C05458=1063.353,412.213,382.958,175.388,37.481,157.115
C05459=1063.360,412.459,382.914,175.394,37.490,157.117
C05460=1063.368,412.705,382.870,175.401,37.500,157.119
C05461=1063.377,412.951,382.826,175.409,37.509,157.122
C05462=1063.386,413.197,382.781,175.416,37.519,157.124
C05463=1063.394,413.443,382.737,175.423,37.528,157.127
C05464=1063.402,413.689,382.693,175.429,37.537,157.129
C05465=1063.411,413.935,382.648,175.436,37.547,157.131
C05466=1063.419,414.181,382.604,175.444,37.556,157.134
C05467=1063.427,414.426,382.559,175.451,37.566,157.136
C05468=1063.438,414.737,382.503,175.459,37.578,157.140
C05469=1063.448,415.046,382.447,175.468,37.590,157.143
C05470=1063.459,415.356,382.391,175.478,37.602,157.146
C05471=1063.469,415.665,382.334,175.486,37.614,157.149
C05472=1063.477,415.911,382.289,175.494,37.624,157.152
C05473=1063.486,416.157,382.245,175.501,37.634,157.154
C05474=1063.494,416.402,382.200,175.508,37.643,157.157
C05475=1063.503,416.648,382.155,175.516,37.653,157.159
C05476=1063.511,416.894,382.110,175.523,37.663,157.162
C05477=1063.520,417.140,382.066,175.530,37.673,157.164
C05478=1063.528,417.385,382.021,175.538,37.683,157.167
C05479=1063.537,417.632,381.976,175.545,37.692,157.170
C05480=1063.545,417.877,381.931,175.553,37.702,157.172
C05481=1063.553,418.123,381.885,175.560,37.712,157.175
C05482=1063.561,418.369,381.840,175.567,37.722,157.177
C05483=1063.570,418.614,381.795,175.575,37.732,157.180
C05484=1063.579,418.860,381.750,175.582,37.742,157.183
C05485=1063.587,419.106,381.705,175.590,37.752,157.185
C05486=1063.596,419.352,381.660,175.597,37.762,157.188
C05487=1063.605,419.597,381.615,175.605,37.772,157.191
C05488=1063.613,419.843,381.569,175.612,37.782,157.193
C05489=1063.622,420.089,381.523,175.620,37.792,157.196
C05490=1063.631,420.335,381.478,175.627,37.803,157.199
C05491=1063.640,420.581,381.433,175.635,37.813,157.201
C05492=1063.648,420.826,381.387,175.643,37.823,157.204
C05493=1063.657,421.072,381.341,175.650,37.833,157.207
C05494=1063.665,421.318,381.296,175.658,37.843,157.210
C05495=1063.673,421.563,381.250,175.665,37.854,157.212
C05496=1063.682,421.808,381.204,175.674,37.864,157.215
C05497=1063.691,422.054,381.158,175.681,37.875,157.218
C05498=1063.700,422.300,381.113,175.689,37.885,157.221
C05499=1063.708,422.546,381.066,175.697,37.896,157.224
C05500=1063.717,422.791,381.021,175.704,37.906,157.226
C05501=1063.726,423.037,380.976,175.713,37.917,157.229
C05502=1063.734,423.282,380.929,175.721,37.927,157.232
C05503=1063.743,423.528,380.883,175.728,37.938,157.235
C05504=1063.752,423.774,380.837,175.736,37.948,157.238
C05505=1063.761,424.019,380.791,175.745,37.959,157.241
C05506=1063.769,424.265,380.745,175.753,37.970,157.244
C05507=1063.778,424.510,380.698,175.760,37.981,157.246
C05508=1063.787,424.756,380.652,175.768,37.991,157.249
C05509=1063.796,425.001,380.606,175.777,38.002,157.252
C05510=1063.804,425.247,380.560,175.785,38.013,157.255
C05511=1063.814,425.492,380.513,175.793,38.024,157.258
C05512=1063.822,425.738,380.467,175.801,38.034,157.261
C05513=1063.832,425.983,380.421,175.809,38.045,157.264
C05514=1063.840,426.229,380.375,175.817,38.056,157.267
C05515=1063.849,426.474,380.328,175.826,38.067,157.270
C05516=1063.858,426.720,380.282,175.834,38.078,157.273
C05517=1063.868,426.966,380.235,175.843,38.089,157.276
C05518=1063.876,427.211,380.188,175.851,38.100,157.279
C05519=1063.885,427.456,380.141,175.860,38.111,157.282
C05520=1063.893,427.702,380.094,175.868,38.122,157.285
C05521=1063.903,427.947,380.048,175.875,38.134,157.288
C05522=1063.912,428.192,380.001,175.884,38.145,157.291
C05523=1063.921,428.438,379.954,175.893,38.156,157.294
C05524=1063.933,428.768,379.890,175.904,38.171,157.298
C05525=1063.945,429.097,379.828,175.916,38.186,157.302
C05526=1063.957,429.427,379.764,175.928,38.202,157.307
C05527=1063.969,429.757,379.701,175.939,38.217,157.311
C05528=1063.978,430.001,379.654,175.948,38.229,157.314
C05529=1063.988,430.247,379.607,175.956,38.240,157.317
C05530=1063.996,430.492,379.560,175.965,38.251,157.320
C05531=1064.006,430.738,379.512,175.974,38.263,157.323
C05532=1064.015,430.983,379.464,175.982,38.274,157.327
C05533=1064.023,431.228,379.418,175.992,38.286,157.330
C05534=1064.033,431.474,379.370,176.001,38.298,157.333
C05535=1064.042,431.719,379.322,176.009,38.310,157.336
C05536=1064.051,431.964,379.275,176.018,38.322,157.340
C05537=1064.060,432.209,379.227,176.027,38.334,157.343
C05538=1064.069,432.455,379.179,176.036,38.345,157.346
C05539=1064.078,432.700,379.132,176.045,38.357,157.350
C05540=1064.088,432.945,379.083,176.054,38.369,157.353
C05541=1064.097,433.190,379.036,176.063,38.381,157.356
C05542=1064.106,433.435,378.988,176.072,38.393,157.359
C05543=1064.116,433.681,378.940,176.082,38.405,157.363
C05544=1064.125,433.925,378.892,176.090,38.417,157.366
C05545=1064.134,434.171,378.844,176.099,38.429,157.369
C05546=1064.144,434.416,378.797,176.109,38.441,157.373
C05547=1064.153,434.660,378.748,176.118,38.454,157.376
C05548=1064.162,434.906,378.701,176.128,38.466,157.380
C05549=1064.172,435.151,378.652,176.137,38.478,157.383
C05550=1064.180,435.396,378.604,176.146,38.490,157.387
C05551=1064.190,435.641,378.556,176.156,38.503,157.390
C05552=1064.200,435.886,378.507,176.165,38.515,157.394
C05553=1064.209,436.132,378.459,176.175,38.527,157.397
C05554=1064.219,436.377,378.411,176.184,38.539,157.400
C05555=1064.229,436.622,378.362,176.194,38.552,157.404
C05556=1064.239,436.867,378.314,176.203,38.564,157.407
C05557=1064.248,437.112,378.265,176.213,38.577,157.411
C05558=1064.257,437.356,378.216,176.223,38.590,157.415
C05559=1064.266,437.601,378.168,176.232,38.602,157.418
C05560=1064.277,437.847,378.119,176.242,38.615,157.422
C05561=1064.287,438.092,378.070,176.251,38.627,157.425
C05562=1064.296,438.337,378.022,176.261,38.640,157.429
C05563=1064.305,438.582,377.973,176.272,38.653,157.433
C05564=1064.315,438.826,377.924,176.281,38.666,157.436
C05565=1064.325,439.071,377.875,176.291,38.679,157.440
C05566=1064.334,439.317,377.826,176.301,38.692,157.444
C05567=1064.344,439.561,377.777,176.310,38.705,157.447
C05568=1064.353,439.806,377.727,176.321,38.718,157.451
C05569=1064.363,440.051,377.678,176.331,38.731,157.455
C05570=1064.373,440.296,377.630,176.341,38.743,157.458
C05571=1064.383,440.541,377.580,176.352,38.757,157.462
C05572=1064.393,440.786,377.531,176.361,38.770,157.466
C05573=1064.402,441.031,377.481,176.372,38.783,157.470
C05574=1064.412,441.275,377.432,176.382,38.797,157.474
C05575=1064.422,441.520,377.382,176.392,38.810,157.477
C05576=1064.432,441.765,377.332,176.403,38.823,157.481
C05577=1064.441,442.010,377.283,176.413,38.836,157.485
C05578=1064.451,442.254,377.234,176.424,38.850,157.489
C05579=1064.461,442.500,377.184,176.434,38.864,157.493
C05580=1064.477,442.869,377.108,176.449,38.884,157.499
C05581=1064.491,443.240,377.033,176.466,38.904,157.505
C05582=1064.507,443.611,376.957,176.482,38.925,157.511
C05583=1064.522,443.980,376.881,176.498,38.946,157.517
C05584=1064.532,444.225,376.832,176.508,38.960,157.521
C05585=1064.542,444.470,376.782,176.519,38.974,157.525
C05586=1064.551,444.714,376.731,176.531,38.987,157.529
C05587=1064.562,444.959,376.682,176.542,39.001,157.533
C05588=1064.572,445.204,376.631,176.552,39.015,157.537
C05589=1064.582,445.448,376.580,176.563,39.029,157.541
C05590=1064.592,445.693,376.531,176.574,39.043,157.545
C05591=1064.603,445.938,376.480,176.586,39.057,157.549
C05592=1064.612,446.182,376.429,176.597,39.072,157.554
C05593=1064.623,446.427,376.378,176.607,39.086,157.558
C05594=1064.633,446.671,376.328,176.619,39.100,157.562
C05595=1064.644,446.916,376.277,176.630,39.114,157.566
C05596=1064.653,447.160,376.226,176.641,39.129,157.570
C05597=1064.664,447.403,376.176,176.653,39.143,157.575
C05598=1064.674,447.647,376.126,176.664,39.158,157.579
C05599=1064.685,447.891,376.075,176.676,39.172,157.583
C05600=1064.697,448.135,376.026,176.687,39.186,157.587
C05601=1064.710,448.379,375.977,176.699,39.199,157.591
C05602=1064.724,448.624,375.929,176.710,39.213,157.595
C05603=1064.739,448.868,375.882,176.722,39.226,157.599
C05604=1064.755,449.113,375.834,176.734,39.238,157.603
C05605=1064.773,449.358,375.788,176.746,39.251,157.607
C05606=1064.791,449.603,375.742,176.758,39.263,157.610
C05607=1064.810,449.849,375.697,176.768,39.275,157.614
C05608=1064.471,449.855,375.431,176.760,39.399,157.648
C05609=1064.452,449.610,375.475,176.748,39.387,157.644
C05610=1064.434,449.364,375.521,176.737,39.375,157.640
C05611=1064.417,449.119,375.566,176.725,39.362,157.637
C05612=1064.401,448.875,375.613,176.713,39.350,157.633
C05613=1064.386,448.629,375.661,176.701,39.337,157.629
C05614=1064.371,448.385,375.710,176.689,39.324,157.625
C05615=1064.358,448.141,375.758,176.678,39.310,157.621
C05616=1064.345,447.897,375.807,176.666,39.296,157.617
C05617=1064.334,447.653,375.858,176.654,39.282,157.612
C05618=1064.324,447.409,375.908,176.643,39.268,157.608
C05619=1064.313,447.165,375.959,176.631,39.254,157.604
C05620=1064.303,446.921,376.009,176.620,39.240,157.600
C05621=1064.293,446.677,376.060,176.609,39.225,157.595
C05622=1064.283,446.433,376.111,176.597,39.211,157.591
C05623=1064.272,446.188,376.161,176.586,39.197,157.587
C05624=1064.262,445.943,376.212,176.575,39.183,157.583
C05625=1064.252,445.699,376.263,176.564,39.169,157.579
C05626=1064.242,445.455,376.313,176.553,39.155,157.575
C05627=1064.231,445.210,376.364,176.542,39.141,157.571
C05628=1064.221,444.965,376.414,176.531,39.127,157.566
C05629=1064.211,444.721,376.464,176.519,39.113,157.562
C05630=1064.201,444.476,376.514,176.508,39.099,157.558
C05631=1064.190,444.231,376.565,176.498,39.085,157.554
C05632=1064.181,443.986,376.615,176.487,39.071,157.550
C05633=1064.167,443.636,376.687,176.472,39.052,157.544
C05634=1064.152,443.284,376.759,176.456,39.032,157.539
C05635=1064.138,442.934,376.830,176.441,39.012,157.533
C05636=1064.123,442.583,376.902,176.425,38.993,157.527
C05637=1064.113,442.337,376.952,176.414,38.980,157.523
C05638=1064.103,442.093,377.001,176.404,38.967,157.520
C05639=1064.094,441.848,377.051,176.394,38.953,157.516
C05640=1064.083,441.603,377.100,176.384,38.940,157.512
C05641=1064.074,441.358,377.150,176.373,38.926,157.508
C05642=1064.064,441.114,377.200,176.363,38.913,157.504
C05643=1064.055,440.869,377.249,176.352,38.900,157.500
C05644=1064.044,440.624,377.298,176.342,38.887,157.497
C05645=1064.035,440.379,377.348,176.332,38.874,157.493
C05646=1064.025,440.135,377.397,176.321,38.861,157.489
C05647=1064.016,439.890,377.446,176.312,38.847,157.485
C05648=1064.005,439.644,377.496,176.302,38.835,157.482
C05649=1063.995,439.399,377.545,176.291,38.822,157.478
C05650=1063.986,439.155,377.594,176.281,38.809,157.474
C05651=1063.976,438.910,377.643,176.272,38.796,157.470
C05652=1063.966,438.665,377.691,176.261,38.783,157.467
C05653=1063.957,438.420,377.741,176.251,38.770,157.463
C05654=1063.947,438.175,377.790,176.242,38.758,157.460
C05655=1063.938,437.930,377.838,176.232,38.745,157.456
C05656=1063.928,437.685,377.887,176.221,38.732,157.452
C05657=1063.919,437.440,377.936,176.212,38.720,157.449
C05658=1063.909,437.195,377.985,176.202,38.707,157.445
C05659=1063.899,436.950,378.033,176.193,38.695,157.442
C05660=1063.890,436.705,378.082,176.183,38.682,157.438
C05661=1063.880,436.460,378.130,176.173,38.670,157.435
C05662=1063.870,436.215,378.179,176.164,38.658,157.431
C05663=1063.860,435.970,378.227,176.154,38.645,157.428
C05664=1063.851,435.725,378.276,176.145,38.633,157.424
C05665=1063.842,435.479,378.324,176.135,38.620,157.421
C05666=1063.833,435.235,378.372,176.126,38.608,157.417
C05667=1063.823,434.990,378.421,176.117,38.596,157.414
C05668=1063.813,434.744,378.469,176.107,38.584,157.410
C05669=1063.804,434.500,378.517,176.098,38.572,157.407
C05670=1063.795,434.255,378.565,176.088,38.560,157.404
C05671=1063.785,434.010,378.613,176.079,38.547,157.400
C05672=1063.776,433.764,378.661,176.070,38.536,157.397
C05673=1063.767,433.519,378.708,176.060,38.523,157.393
C05674=1063.757,433.274,378.757,176.051,38.512,157.390
C05675=1063.748,433.029,378.805,176.042,38.500,157.387
C05676=1063.739,432.784,378.852,176.032,38.488,157.383
C05677=1063.729,432.538,378.900,176.024,38.476,157.380
C05678=1063.720,432.293,378.947,176.015,38.464,157.377
C05679=1063.711,432.048,378.996,176.006,38.452,157.373
C05680=1063.702,431.803,379.043,175.997,38.440,157.370
C05681=1063.692,431.558,379.091,175.987,38.429,157.367
C05682=1063.683,431.313,379.139,175.979,38.417,157.364
C05683=1063.674,431.067,379.186,175.970,38.405,157.360
C05684=1063.665,430.822,379.233,175.961,38.394,157.357
C05685=1063.656,430.576,379.281,175.953,38.382,157.354
C05686=1063.647,430.331,379.328,175.944,38.371,157.351
C05687=1063.638,430.086,379.376,175.934,38.360,157.348
C05688=1063.629,429.840,379.423,175.925,38.348,157.345
C05689=1063.616,429.509,379.487,175.914,38.332,157.340
C05690=1063.605,429.178,379.550,175.902,38.317,157.336
C05691=1063.592,428.846,379.614,175.891,38.302,157.332
C05692=1063.579,428.514,379.677,175.879,38.287,157.328
C05693=1063.570,428.269,379.725,175.871,38.276,157.325
C05694=1063.562,428.024,379.771,175.862,38.264,157.322
C05695=1063.553,427.778,379.818,175.854,38.253,157.319
C05696=1063.543,427.533,379.865,175.845,38.242,157.315
C05697=1063.535,427.287,379.912,175.837,38.231,157.312
C05698=1063.526,427.042,379.959,175.828,38.220,157.309
C05699=1063.517,426.796,380.005,175.820,38.209,157.306
C05700=1063.508,426.551,380.052,175.811,38.198,157.303
C05701=1063.499,426.305,380.099,175.803,38.187,157.300
C05702=1063.490,426.060,380.145,175.794,38.176,157.297
C05703=1063.481,425.814,380.191,175.787,38.165,157.294
C05704=1063.472,425.569,380.238,175.779,38.154,157.292
C05705=1063.463,425.323,380.284,175.770,38.144,157.289
C05706=1063.454,425.078,380.330,175.762,38.133,157.286
C05707=1063.446,424.833,380.377,175.753,38.122,157.283
C05708=1063.437,424.587,380.423,175.745,38.111,157.280
C05709=1063.428,424.341,380.469,175.738,38.100,157.277
C05710=1063.419,424.096,380.515,175.729,38.090,157.274
C05711=1063.410,423.850,380.561,175.721,38.079,157.271
C05712=1063.401,423.605,380.608,175.713,38.069,157.268
C05713=1063.392,423.360,380.654,175.706,38.058,157.265
C05714=1063.384,423.113,380.700,175.697,38.047,157.263
C05715=1063.374,422.868,380.746,175.689,38.037,157.260
C05716=1063.366,422.622,380.792,175.682,38.027,157.257
C05717=1063.357,422.376,380.837,175.673,38.016,157.254
C05718=1063.349,422.131,380.884,175.665,38.006,157.251
C05719=1063.340,421.886,380.929,175.658,37.995,157.248
C05720=1063.331,421.640,380.975,175.650,37.985,157.246
C05721=1063.323,421.394,381.021,175.643,37.975,157.243
C05722=1063.314,421.149,381.067,175.634,37.964,157.240
C05723=1063.306,420.903,381.112,175.626,37.954,157.237
C05724=1063.297,420.657,381.158,175.619,37.944,157.235
C05725=1063.288,420.411,381.203,175.611,37.934,157.232
C05726=1063.280,420.165,381.249,175.604,37.924,157.229
C05727=1063.272,419.920,381.294,175.596,37.913,157.227
C05728=1063.263,419.674,381.340,175.589,37.903,157.224
C05729=1063.254,419.429,381.385,175.580,37.893,157.221
C05730=1063.245,419.183,381.430,175.573,37.883,157.219
C05731=1063.236,418.938,381.476,175.565,37.873,157.216
C05732=1063.228,418.691,381.522,175.558,37.863,157.213
C05733=1063.220,418.446,381.566,175.550,37.853,157.210
C05734=1063.211,418.200,381.611,175.543,37.844,157.208
C05735=1063.202,417.954,381.657,175.535,37.834,157.205
C05736=1063.194,417.709,381.702,175.528,37.824,157.203
C05737=1063.185,417.462,381.746,175.520,37.814,157.200
C05738=1063.177,417.217,381.792,175.513,37.804,157.197
C05739=1063.168,416.971,381.836,175.506,37.794,157.195
C05740=1063.160,416.725,381.882,175.498,37.784,157.192
C05741=1063.152,416.479,381.927,175.491,37.775,157.190
C05742=1063.143,416.234,381.972,175.484,37.765,157.187
C05743=1063.135,415.987,382.016,175.476,37.755,157.185
C05744=1063.126,415.742,382.061,175.469,37.745,157.182
C05745=1063.115,415.431,382.118,175.460,37.733,157.179
C05746=1063.104,415.119,382.175,175.451,37.721,157.176
C05747=1063.095,414.808,382.231,175.442,37.709,157.172
C05748=1063.084,414.496,382.288,175.432,37.697,157.169
C05749=1063.076,414.251,382.332,175.426,37.687,157.167
C05750=1063.067,414.004,382.377,175.419,37.678,157.164
C05751=1063.059,413.759,382.421,175.411,37.668,157.162
C05752=1063.051,413.513,382.465,175.404,37.659,157.159
C05753=1063.042,413.267,382.510,175.397,37.650,157.157
C05754=1063.034,413.021,382.554,175.390,37.640,157.154
C05755=1063.025,412.775,382.598,175.384,37.631,157.152
C05756=1063.016,412.529,382.642,175.376,37.622,157.150
C05757=1063.008,412.283,382.687,175.369,37.613,157.147
C05758=1063.000,412.037,382.731,175.362,37.603,157.145
C05759=1062.992,411.792,382.775,175.355,37.594,157.142
C05760=1062.983,411.545,382.819,175.349,37.585,157.140
C05761=1062.975,411.299,382.863,175.342,37.576,157.138
C05762=1062.967,411.053,382.907,175.335,37.567,157.135
C05763=1062.958,410.807,382.950,175.327,37.558,157.133
C05764=1062.950,410.562,382.995,175.321,37.549,157.131
C05765=1062.942,410.316,383.039,175.314,37.540,157.128
C05766=1062.934,410.070,383.083,175.307,37.531,157.126
C05767=1062.926,409.824,383.126,175.300,37.522,157.124
C05768=1062.917,409.577,383.170,175.294,37.513,157.121
C05769=1062.909,409.331,383.215,175.287,37.504,157.119
C05770=1062.901,409.085,383.258,175.280,37.495,157.117
C05771=1062.893,408.839,383.301,175.274,37.486,157.114
C05772=1062.885,408.593,383.346,175.267,37.477,157.112
C05773=1062.876,408.347,383.389,175.260,37.468,157.110
C05774=1062.869,408.101,383.432,175.254,37.459,157.107
C05775=1062.861,407.856,383.476,175.247,37.450,157.105
C05776=1062.853,407.610,383.519,175.240,37.441,157.103
C05777=1062.845,407.363,383.563,175.234,37.432,157.101
C05778=1062.837,407.117,383.607,175.227,37.424,157.098
C05779=1062.829,406.871,383.650,175.220,37.415,157.096
C05780=1062.821,406.625,383.694,175.214,37.406,157.094
C05781=1062.813,406.379,383.738,175.208,37.398,157.092
C05782=1062.805,406.133,383.780,175.202,37.389,157.089
C05783=1062.797,405.887,383.824,175.195,37.380,157.087
C05784=1062.789,405.641,383.867,175.188,37.372,157.085
C05785=1062.781,405.395,383.911,175.182,37.363,157.083
C05786=1062.773,405.148,383.953,175.175,37.355,157.081
C05787=1062.765,404.902,383.997,175.169,37.346,157.078
C05788=1062.757,404.656,384.039,175.162,37.337,157.076
C05789=1062.749,404.410,384.083,175.157,37.329,157.074
C05790=1062.741,404.164,384.126,175.150,37.320,157.072
C05791=1062.734,403.917,384.168,175.144,37.312,157.070
C05792=1062.725,403.671,384.211,175.137,37.303,157.068
C05793=1062.717,403.425,384.254,175.131,37.295,157.066
C05794=1062.709,403.178,384.297,175.125,37.287,157.063
C05795=1062.702,402.933,384.340,175.119,37.279,157.061
C05796=1062.693,402.687,384.383,175.112,37.270,157.059
C05797=1062.686,402.440,384.426,175.106,37.261,157.057
C05798=1062.678,402.195,384.469,175.099,37.253,157.055
C05799=1062.669,401.948,384.511,175.094,37.245,157.053
C05800=1062.661,401.702,384.554,175.087,37.237,157.051
C05801=1062.652,401.395,384.606,175.079,37.227,157.048
C05802=1062.642,401.089,384.659,175.072,37.216,157.046
C05803=1062.632,400.783,384.713,175.064,37.206,157.043
C05804=1062.622,400.476,384.765,175.056,37.196,157.040
C05805=1062.615,400.230,384.807,175.051,37.188,157.038
C05806=1062.606,399.984,384.850,175.044,37.180,157.036
C05807=1062.599,399.738,384.893,175.038,37.172,157.034
C05808=1062.591,399.491,384.935,175.033,37.164,157.032
C05809=1062.584,399.245,384.977,175.026,37.156,157.030
C05810=1062.575,398.999,385.019,175.020,37.148,157.028
C05811=1062.568,398.753,385.061,175.014,37.140,157.026
C05812=1062.560,398.506,385.104,175.008,37.132,157.024
C05813=1062.552,398.261,385.146,175.002,37.124,157.022
C05814=1062.545,398.014,385.189,174.996,37.116,157.020
C05815=1062.537,397.768,385.231,174.990,37.108,157.018
C05816=1062.529,397.521,385.272,174.985,37.100,157.016
C05817=1062.522,397.275,385.314,174.978,37.092,157.014
C05818=1062.513,397.028,385.357,174.972,37.085,157.012
C05819=1062.506,396.782,385.398,174.967,37.077,157.010
C05820=1062.498,396.537,385.440,174.960,37.069,157.009
C05821=1062.490,396.290,385.483,174.955,37.061,157.007
C05822=1062.483,396.043,385.524,174.949,37.053,157.005
C05823=1062.474,395.798,385.565,174.943,37.046,157.003
C05824=1062.467,395.552,385.607,174.937,37.038,157.001
C05825=1062.459,395.305,385.650,174.931,37.030,156.999
C05826=1062.451,395.058,385.691,174.926,37.023,156.997
C05827=1062.444,394.812,385.733,174.919,37.014,156.995
C05828=1062.436,394.566,385.775,174.914,37.007,156.993
C05829=1062.428,394.319,385.816,174.908,36.999,156.991
C05830=1062.421,394.073,385.858,174.902,36.992,156.989
C05831=1062.413,393.827,385.899,174.896,36.984,156.987
C05832=1062.406,393.581,385.941,174.891,36.977,156.986
C05833=1062.398,393.334,385.982,174.885,36.969,156.984
C05834=1062.391,393.088,386.023,174.880,36.961,156.982
C05835=1062.383,392.842,386.065,174.873,36.954,156.980
C05836=1062.376,392.595,386.106,174.868,36.946,156.978
C05837=1062.367,392.349,386.148,174.862,36.939,156.976
C05838=1062.359,392.102,386.189,174.857,36.932,156.974
C05839=1062.352,391.856,386.231,174.850,36.924,156.973
C05840=1062.345,391.609,386.272,174.845,36.916,156.971
C05841=1062.337,391.363,386.313,174.840,36.909,156.969
C05842=1062.329,391.117,386.354,174.834,36.902,156.967
C05843=1062.322,390.870,386.396,174.829,36.895,156.965
C05844=1062.314,390.624,386.436,174.823,36.887,156.963
C05845=1062.307,390.377,386.478,174.817,36.880,156.962
C05846=1062.299,390.131,386.519,174.811,36.872,156.960
C05847=1062.291,389.884,386.559,174.806,36.865,156.958
C05848=1062.284,389.638,386.601,174.801,36.858,156.956
C05849=1062.276,389.391,386.641,174.795,36.851,156.955
C05850=1062.269,389.145,386.682,174.790,36.844,156.953
C05851=1062.261,388.899,386.723,174.784,36.836,156.951
C05852=1062.254,388.653,386.764,174.778,36.829,156.949
C05853=1062.246,388.406,386.805,174.773,36.822,156.947
C05854=1062.239,388.160,386.846,174.767,36.815,156.946
C05855=1062.231,387.914,386.886,174.762,36.808,156.944
C05856=1062.223,387.667,386.926,174.757,36.801,156.942
C05857=1062.214,387.377,386.975,174.751,36.792,156.940
C05858=1062.205,387.088,387.023,174.743,36.784,156.938
C05859=1062.196,386.798,387.070,174.737,36.775,156.936
C05860=1062.188,386.508,387.118,174.731,36.767,156.934
C05861=1062.180,386.262,387.159,174.726,36.760,156.932
C05862=1062.173,386.015,387.199,174.721,36.753,156.931
C05863=1062.165,385.769,387.240,174.714,36.746,156.929
C05864=1062.158,385.522,387.280,174.709,36.739,156.927
C05865=1062.150,385.275,387.321,174.704,36.732,156.926
C05866=1062.143,385.029,387.360,174.699,36.725,156.924
C05867=1062.136,384.783,387.402,174.693,36.718,156.922
C05868=1062.128,384.536,387.441,174.688,36.712,156.921
C05869=1062.120,384.289,387.482,174.683,36.704,156.919
C05870=1062.114,384.043,387.522,174.678,36.697,156.917
C05871=1062.106,383.796,387.562,174.672,36.691,156.916
C05872=1062.099,383.549,387.603,174.667,36.684,156.914
C05873=1062.092,383.303,387.643,174.662,36.677,156.912
C05874=1062.084,383.056,387.683,174.657,36.670,156.911
C05875=1062.077,382.810,387.724,174.651,36.663,156.909
C05876=1062.070,382.564,387.764,174.646,36.656,156.907
C05877=1062.062,382.317,387.804,174.641,36.650,156.906
C05878=1062.056,382.070,387.844,174.636,36.643,156.904
C05879=1062.048,381.824,387.884,174.631,36.636,156.902
C05880=1062.040,381.578,387.924,174.626,36.629,156.901
C05881=1062.033,381.330,387.964,174.620,36.622,156.899
C05882=1062.026,381.084,388.004,174.615,36.616,156.897
C05883=1062.019,380.837,388.044,174.610,36.609,156.896
C05884=1062.011,380.591,388.083,174.605,36.602,156.894
C05885=1062.004,380.344,388.124,174.600,36.596,156.893
C05886=1061.997,380.097,388.164,174.595,36.589,156.891
C05887=1061.990,379.851,388.203,174.589,36.583,156.890
C05888=1061.982,379.604,388.243,174.584,36.576,156.888
C05889=1061.975,379.358,388.283,174.579,36.569,156.886
C05890=1061.967,379.111,388.323,174.574,36.563,156.885
C05891=1061.960,378.864,388.362,174.569,36.556,156.883
C05892=1061.953,378.617,388.402,174.564,36.550,156.882
C05893=1061.945,378.371,388.441,174.559,36.543,156.880
C05894=1061.938,378.124,388.481,174.553,36.536,156.878
C05895=1061.931,377.877,388.520,174.549,36.530,156.877
C05896=1061.923,377.630,388.560,174.544,36.524,156.875
C05897=1061.916,377.384,388.599,174.539,36.517,156.874
C05898=1061.909,377.137,388.638,174.534,36.511,156.872
C05899=1061.902,376.890,388.678,174.529,36.504,156.871
C05900=1061.894,376.644,388.718,174.524,36.498,156.869
C05901=1061.887,376.397,388.757,174.519,36.491,156.868
C05902=1061.880,376.150,388.796,174.514,36.485,156.866
C05903=1061.873,375.904,388.835,174.509,36.479,156.865
C05904=1061.865,375.657,388.875,174.504,36.472,156.863
C05905=1061.859,375.410,388.914,174.499,36.466,156.862
C05906=1061.851,375.164,388.954,174.495,36.459,156.860
C05907=1061.844,374.916,388.993,174.490,36.453,156.859
C05908=1061.837,374.670,389.032,174.485,36.446,156.857
C05909=1061.830,374.423,389.071,174.480,36.440,156.856
C05910=1061.823,374.176,389.110,174.475,36.434,156.854
C05911=1061.816,373.929,389.150,174.470,36.428,156.853
C05912=1061.809,373.682,389.189,174.465,36.422,156.851
C05913=1061.801,373.423,389.229,174.459,36.415,156.850
C05914=1061.794,373.166,389.271,174.455,36.408,156.848
C05915=1061.786,372.907,389.311,174.450,36.402,156.846
C05916=1061.779,372.648,389.352,174.445,36.395,156.845
C05917=1061.773,372.411,389.389,174.440,36.389,156.843
C05918=1061.765,372.175,389.427,174.435,36.383,156.842
C05919=1061.758,371.938,389.464,174.431,36.377,156.841
C05920=1061.751,371.701,389.501,174.427,36.372,156.839
C05921=1061.744,371.455,389.539,174.422,36.365,156.838
C05922=1061.737,371.208,389.578,174.417,36.359,156.836
C05923=1061.730,370.962,389.618,174.412,36.353,156.835
C05924=1061.722,370.715,389.656,174.407,36.347,156.834
C05925=1061.715,370.467,389.695,174.402,36.341,156.832
C05926=1061.708,370.220,389.733,174.398,36.335,156.831
C05927=1061.701,369.974,389.772,174.393,36.329,156.829
C05928=1061.694,369.727,389.810,174.388,36.323,156.828
C05929=1061.687,369.480,389.849,174.383,36.317,156.827
C05930=1061.680,369.234,389.888,174.378,36.311,156.825
C05931=1061.673,368.987,389.926,174.374,36.305,156.824
C05932=1061.665,368.740,389.965,174.369,36.298,156.822
C05933=1061.659,368.493,390.003,174.365,36.293,156.821
C05934=1061.651,368.246,390.041,174.360,36.287,156.820
C05935=1061.644,367.999,390.080,174.355,36.281,156.818
C05936=1061.637,367.752,390.119,174.351,36.274,156.817
C05937=1061.630,367.505,390.157,174.346,36.269,156.815
C05938=1061.623,367.258,390.195,174.341,36.263,156.814
C05939=1061.615,367.011,390.234,174.336,36.257,156.812
C05940=1061.609,366.764,390.272,174.332,36.251,156.811
C05941=1061.602,366.517,390.311,174.328,36.245,156.810
C05942=1061.595,366.270,390.348,174.323,36.239,156.808
C05943=1061.588,366.023,390.387,174.318,36.233,156.807
C05944=1061.581,365.776,390.424,174.313,36.227,156.806
C05945=1061.575,365.530,390.463,174.309,36.222,156.804
C05946=1061.567,365.283,390.500,174.304,36.215,156.803
C05947=1061.561,365.036,390.539,174.300,36.210,156.802
C05948=1061.554,364.789,390.577,174.295,36.204,156.800
C05949=1061.547,364.542,390.616,174.291,36.198,156.799
C05950=1061.540,364.295,390.654,174.286,36.192,156.797
C05951=1061.532,364.048,390.692,174.281,36.186,156.796
C05952=1061.525,363.801,390.730,174.277,36.181,156.795
C05953=1061.519,363.554,390.768,174.273,36.175,156.793
C05954=1061.511,363.306,390.805,174.268,36.169,156.792
C05955=1061.505,363.061,390.843,174.263,36.163,156.791
C05956=1061.498,362.813,390.881,174.259,36.158,156.790
C05957=1061.491,362.566,390.919,174.255,36.152,156.788
C05958=1061.484,362.319,390.956,174.250,36.146,156.787
C05959=1061.477,362.071,390.994,174.245,36.140,156.786
C05960=1061.469,361.825,391.033,174.241,36.135,156.784
C05961=1061.462,361.578,391.070,174.237,36.129,156.783
C05962=1061.456,361.331,391.108,174.232,36.124,156.782
C05963=1061.449,361.084,391.145,174.228,36.118,156.780
C05964=1061.442,360.837,391.183,174.223,36.112,156.779
C05965=1061.435,360.590,391.220,174.219,36.107,156.778
C05966=1061.427,360.343,391.258,174.215,36.101,156.777
C05967=1061.421,360.096,391.296,174.210,36.096,156.775
C05968=1061.414,359.849,391.333,174.205,36.090,156.774
C05969=1061.407,359.597,391.372,174.202,36.084,156.773
C05970=1061.400,359.347,391.409,174.197,36.079,156.771
C05971=1061.393,359.095,391.448,174.192,36.073,156.770
C05972=1061.386,358.845,391.486,174.187,36.067,156.769
C05973=1061.379,358.597,391.523,174.184,36.062,156.768
C05974=1061.372,358.350,391.560,174.179,36.056,156.766
C05975=1061.365,358.103,391.598,174.174,36.051,156.765
C05976=1061.358,357.857,391.635,174.171,36.045,156.764
C05977=1061.351,357.609,391.672,174.166,36.039,156.762
C05978=1061.345,357.361,391.710,174.161,36.034,156.761
C05979=1061.338,357.115,391.747,174.157,36.029,156.760
C05980=1061.331,356.868,391.785,174.153,36.023,156.759
C05981=1061.324,356.620,391.821,174.148,36.018,156.758
C05982=1061.317,356.374,391.859,174.144,36.012,156.756
C05983=1061.310,356.126,391.896,174.140,36.007,156.755
C05984=1061.303,355.879,391.933,174.136,36.002,156.754
C05985=1061.296,355.632,391.970,174.131,35.996,156.752
C05986=1061.290,355.385,392.007,174.127,35.991,156.751
C05987=1061.283,355.138,392.044,174.123,35.985,156.750
C05988=1061.276,354.890,392.081,174.119,35.980,156.749
C05989=1061.269,354.643,392.118,174.114,35.975,156.748
C05990=1061.262,354.396,392.155,174.110,35.969,156.746
C05991=1061.255,354.149,392.192,174.106,35.964,156.745
C05992=1061.249,353.902,392.229,174.101,35.958,156.744
C05993=1061.242,353.655,392.266,174.097,35.953,156.743
C05994=1061.235,353.408,392.303,174.093,35.948,156.741
C05995=1061.228,353.160,392.340,174.089,35.943,156.740
C05996=1061.222,352.914,392.377,174.085,35.937,156.739
C05997=1061.215,352.666,392.413,174.080,35.932,156.738
C05998=1061.208,352.419,392.449,174.076,35.927,156.737
C05999=1061.200,352.172,392.487,174.072,35.921,156.735
C06000=1061.194,351.925,392.523,174.068,35.916,156.734
C06001=1061.187,351.677,392.560,174.064,35.910,156.733
C06002=1061.181,351.430,392.597,174.059,35.905,156.732
C06003=1061.174,351.182,392.633,174.056,35.900,156.731
C06004=1061.167,350.936,392.671,174.051,35.895,156.730
C06005=1061.160,350.688,392.707,174.047,35.890,156.728
C06006=1061.153,350.441,392.743,174.043,35.884,156.727
C06007=1061.146,350.194,392.780,174.038,35.879,156.726
C06008=1061.140,349.947,392.816,174.035,35.874,156.725
C06009=1061.132,349.699,392.853,174.030,35.869,156.724
C06010=1061.126,349.452,392.889,174.027,35.864,156.723
C06011=1061.120,349.205,392.926,174.022,35.859,156.721
C06012=1061.113,348.957,392.962,174.018,35.854,156.720
C06013=1061.106,348.711,392.998,174.014,35.848,156.719
C06014=1061.099,348.463,393.035,174.010,35.843,156.718
C06015=1061.092,348.216,393.071,174.006,35.838,156.717
C06016=1061.085,347.969,393.107,174.002,35.833,156.716
C06017=1061.078,347.721,393.144,173.998,35.828,156.714
C06018=1061.072,347.474,393.181,173.994,35.823,156.713
C06019=1061.066,347.227,393.217,173.989,35.817,156.712
C06020=1061.058,346.979,393.253,173.986,35.812,156.711
C06021=1061.052,346.737,393.288,173.981,35.807,156.710
C06022=1061.045,346.497,393.323,173.978,35.803,156.709
C06023=1061.039,346.254,393.359,173.973,35.798,156.708
C06024=1061.032,346.013,393.394,173.970,35.792,156.707
C06025=1061.026,345.771,393.430,173.966,35.788,156.706
C06026=1061.019,345.529,393.465,173.962,35.783,156.704
C06027=1061.012,345.288,393.500,173.958,35.778,156.703
C06028=1061.006,345.046,393.535,173.954,35.773,156.702
C06029=1061.000,344.799,393.572,173.950,35.768,156.701
C06030=1060.993,344.552,393.607,173.946,35.763,156.700
C06031=1060.986,344.303,393.644,173.942,35.758,156.699
C06032=1060.979,344.057,393.679,173.938,35.753,156.698
C06033=1060.973,343.809,393.715,173.934,35.748,156.697
C06034=1060.966,343.562,393.751,173.930,35.743,156.696
C06035=1060.960,343.315,393.787,173.926,35.738,156.694
C06036=1060.952,343.067,393.823,173.922,35.733,156.693
C06037=1060.946,342.819,393.859,173.918,35.728,156.692
C06038=1060.939,342.573,393.894,173.914,35.723,156.691
C06039=1060.932,342.325,393.930,173.911,35.718,156.690
C06040=1060.926,342.078,393.966,173.906,35.713,156.689
C06041=1060.919,341.830,394.002,173.903,35.708,156.688
C06042=1060.913,341.583,394.037,173.898,35.704,156.687
C06043=1060.905,341.336,394.073,173.895,35.698,156.686
C06044=1060.899,341.088,394.108,173.890,35.693,156.685
C06045=1060.892,340.841,394.145,173.887,35.689,156.684
C06046=1060.886,340.594,394.180,173.883,35.684,156.682
C06047=1060.878,340.346,394.215,173.879,35.679,156.681
C06048=1060.872,340.098,394.251,173.875,35.674,156.680
C06049=1060.865,339.852,394.287,173.872,35.669,156.679
C06050=1060.858,339.604,394.322,173.867,35.664,156.678
C06051=1060.852,339.356,394.358,173.864,35.660,156.677
C06052=1060.846,339.109,394.393,173.859,35.654,156.676
C06053=1060.839,338.862,394.428,173.856,35.650,156.675
C06054=1060.832,338.615,394.465,173.852,35.645,156.674
C06055=1060.826,338.367,394.500,173.848,35.640,156.673
C06056=1060.819,338.120,394.535,173.844,35.636,156.672
C06057=1060.813,337.872,394.571,173.841,35.630,156.671
C06058=1060.806,337.625,394.606,173.836,35.626,156.670
C06059=1060.799,337.378,394.641,173.833,35.621,156.669
C06060=1060.793,337.130,394.676,173.829,35.616,156.668
C06061=1060.787,336.883,394.712,173.825,35.612,156.666
C06062=1060.780,336.635,394.747,173.821,35.606,156.665
C06063=1060.773,336.388,394.782,173.818,35.602,156.664
C06064=1060.766,336.140,394.817,173.813,35.597,156.663
C06065=1060.759,335.893,394.852,173.810,35.593,156.662
C06066=1060.753,335.646,394.887,173.806,35.587,156.661
C06067=1060.746,335.398,394.922,173.802,35.583,156.660
C06068=1060.739,335.150,394.957,173.798,35.578,156.659
C06069=1060.733,334.903,394.992,173.795,35.574,156.658
C06070=1060.727,334.655,395.028,173.791,35.569,156.657
C06071=1060.720,334.408,395.063,173.787,35.564,156.656
C06072=1060.713,334.161,395.098,173.783,35.559,156.655
C06073=1060.707,333.913,395.132,173.780,35.555,156.654
C06074=1060.700,333.665,395.168,173.776,35.550,156.653
C06075=1060.693,333.418,395.203,173.772,35.546,156.652
C06076=1060.686,333.171,395.238,173.769,35.541,156.651
C06077=1060.680,332.926,395.272,173.765,35.536,156.650
C06078=1060.673,332.683,395.306,173.761,35.532,156.649
C06079=1060.667,332.439,395.340,173.757,35.527,156.648
C06080=1060.661,332.195,395.375,173.754,35.523,156.647
C06081=1060.654,331.951,395.409,173.750,35.518,156.646
C06082=1060.648,331.707,395.443,173.747,35.513,156.645
C06083=1060.641,331.462,395.478,173.743,35.509,156.644
C06084=1060.635,331.218,395.512,173.739,35.504,156.643
C06085=1060.629,330.971,395.547,173.736,35.500,156.642
C06086=1060.623,330.723,395.582,173.732,35.495,156.641
C06087=1060.616,330.476,395.617,173.729,35.490,156.640
C06088=1060.609,330.228,395.651,173.724,35.486,156.639
C06089=1060.602,329.981,395.686,173.721,35.481,156.638
C06090=1060.595,329.733,395.720,173.717,35.477,156.637
C06091=1060.588,329.486,395.755,173.714,35.472,156.636
C06092=1060.582,329.239,395.789,173.710,35.468,156.635
C06093=1060.576,328.991,395.823,173.706,35.463,156.634
C06094=1060.568,328.744,395.858,173.703,35.459,156.633
C06095=1060.562,328.496,395.892,173.699,35.454,156.632
C06096=1060.555,328.248,395.926,173.695,35.450,156.631
C06097=1060.548,328.001,395.961,173.692,35.445,156.630
C06098=1060.542,327.753,395.995,173.688,35.441,156.629
C06099=1060.535,327.505,396.029,173.685,35.437,156.628
C06100=1060.528,327.258,396.063,173.681,35.432,156.627
C06101=1060.521,327.010,396.098,173.677,35.427,156.626
C06102=1060.515,326.763,396.132,173.673,35.423,156.625
C06103=1060.508,326.515,396.166,173.670,35.419,156.625
C06104=1060.502,326.267,396.201,173.667,35.414,156.624
C06105=1060.495,326.020,396.235,173.663,35.410,156.623
C06106=1060.489,325.772,396.269,173.659,35.405,156.622
C06107=1060.482,325.525,396.304,173.655,35.401,156.621
C06108=1060.475,325.277,396.338,173.652,35.396,156.620
C06109=1060.469,325.030,396.372,173.649,35.392,156.619
C06110=1060.462,324.782,396.405,173.645,35.388,156.618
C06111=1060.455,324.534,396.440,173.642,35.383,156.617
C06112=1060.449,324.287,396.474,173.638,35.379,156.616
C06113=1060.442,324.039,396.508,173.634,35.374,156.615
C06114=1060.436,323.791,396.542,173.631,35.370,156.614
C06115=1060.429,323.545,396.576,173.627,35.366,156.613
C06116=1060.423,323.297,396.610,173.624,35.361,156.612
C06117=1060.417,323.049,396.644,173.620,35.357,156.611
C06118=1060.410,322.802,396.678,173.617,35.352,156.610
C06119=1060.403,322.554,396.712,173.614,35.348,156.609
C06120=1060.397,322.307,396.746,173.610,35.344,156.608
C06121=1060.390,322.059,396.780,173.606,35.339,156.607
C06122=1060.384,321.811,396.813,173.602,35.335,156.607
C06123=1060.377,321.563,396.847,173.599,35.330,156.606
C06124=1060.371,321.316,396.881,173.596,35.326,156.605
C06125=1060.364,321.068,396.915,173.592,35.322,156.604
C06126=1060.358,320.821,396.949,173.589,35.317,156.603
C06127=1060.351,320.573,396.983,173.585,35.313,156.602
C06128=1060.346,320.325,397.016,173.582,35.308,156.601
C06129=1060.338,320.078,397.050,173.579,35.304,156.600
C06130=1060.333,319.830,397.084,173.575,35.299,156.599
C06131=1060.325,319.583,397.118,173.572,35.295,156.598
C06132=1060.320,319.335,397.152,173.568,35.291,156.597
C06133=1060.313,319.088,397.185,173.564,35.287,156.596
C06134=1060.306,318.841,397.219,173.561,35.282,156.595
C06135=1060.300,318.594,397.253,173.557,35.278,156.594
C06136=1060.294,318.347,397.287,173.554,35.273,156.593
C06137=1060.288,318.101,397.320,173.551,35.269,156.593
C06138=1060.281,317.854,397.353,173.547,35.265,156.592
C06139=1060.275,317.607,397.387,173.544,35.261,156.591
C06140=1060.268,317.360,397.420,173.541,35.256,156.590
C06141=1060.263,317.112,397.453,173.537,35.252,156.589
C06142=1060.256,316.865,397.487,173.534,35.248,156.588
C06143=1060.250,316.617,397.521,173.530,35.243,156.587
C06144=1060.243,316.370,397.554,173.527,35.239,156.586
C06145=1060.238,316.122,397.587,173.524,35.234,156.585
C06146=1060.230,315.874,397.621,173.520,35.230,156.584
C06147=1060.225,315.626,397.655,173.517,35.226,156.583
C06148=1060.218,315.379,397.688,173.514,35.222,156.582
C06149=1060.212,315.130,397.722,173.510,35.217,156.582
C06150=1060.205,314.884,397.755,173.507,35.213,156.581
C06151=1060.199,314.636,397.788,173.504,35.209,156.580
C06152=1060.193,314.389,397.822,173.500,35.205,156.579
C06153=1060.186,314.140,397.855,173.497,35.200,156.578
C06154=1060.181,313.892,397.888,173.493,35.196,156.577
C06155=1060.174,313.645,397.922,173.490,35.191,156.576
C06156=1060.167,313.397,397.955,173.487,35.187,156.575
C06157=1060.161,313.150,397.988,173.483,35.183,156.574
C06158=1060.155,312.902,398.021,173.480,35.179,156.573
C06159=1060.148,312.654,398.054,173.477,35.175,156.573
C06160=1060.141,312.407,398.087,173.473,35.171,156.572
C06161=1060.135,312.159,398.120,173.470,35.167,156.571
C06162=1060.128,311.911,398.153,173.467,35.163,156.570
C06163=1060.122,311.663,398.186,173.463,35.158,156.569
C06164=1060.116,311.416,398.218,173.460,35.154,156.568
C06165=1060.109,311.167,398.252,173.457,35.150,156.567
C06166=1060.102,310.920,398.285,173.453,35.146,156.567
C06167=1060.095,310.673,398.317,173.450,35.142,156.566
C06168=1060.089,310.426,398.350,173.447,35.138,156.565
C06169=1060.082,310.177,398.383,173.443,35.133,156.564
C06170=1060.076,309.930,398.416,173.440,35.129,156.563
C06171=1060.069,309.682,398.448,173.437,35.125,156.562
C06172=1060.063,309.434,398.481,173.433,35.121,156.561
C06173=1060.056,309.186,398.514,173.430,35.117,156.560
C06174=1060.050,308.939,398.547,173.427,35.113,156.560
C06175=1060.043,308.691,398.580,173.424,35.109,156.559
C06176=1060.037,308.443,398.613,173.421,35.105,156.558
C06177=1060.031,308.196,398.645,173.418,35.101,156.557
C06178=1060.023,307.948,398.678,173.414,35.096,156.556
C06179=1060.017,307.700,398.710,173.411,35.092,156.555
C06180=1060.011,307.452,398.743,173.408,35.088,156.554
C06181=1060.005,307.204,398.775,173.404,35.084,156.554
C06182=1059.998,306.957,398.808,173.401,35.080,156.553
C06183=1059.992,306.709,398.841,173.398,35.076,156.552
C06184=1059.986,306.462,398.874,173.395,35.072,156.551
C06185=1059.978,306.214,398.906,173.391,35.068,156.550
C06186=1059.972,305.965,398.938,173.388,35.064,156.549
C06187=1059.966,305.718,398.971,173.385,35.060,156.548
C06188=1059.960,305.470,399.004,173.382,35.055,156.548
C06189=1059.953,305.225,399.036,173.379,35.052,156.547
C06190=1059.947,304.980,399.068,173.376,35.048,156.546
C06191=1059.941,304.736,399.099,173.372,35.044,156.545
C06192=1059.935,304.491,399.132,173.369,35.040,156.544
C06193=1059.928,304.246,399.164,173.366,35.035,156.543
C06194=1059.922,304.001,399.196,173.362,35.031,156.543
C06195=1059.915,303.756,399.228,173.360,35.027,156.542
C06196=1059.910,303.511,399.259,173.357,35.023,156.541
C06197=1059.904,303.264,399.292,173.353,35.020,156.540
C06198=1059.897,303.016,399.325,173.350,35.015,156.539
C06199=1059.891,302.768,399.357,173.347,35.011,156.538
C06200=1059.884,302.520,399.389,173.344,35.007,156.538
C06201=1059.878,302.272,399.421,173.340,35.003,156.537
C06202=1059.872,302.025,399.454,173.338,34.999,156.536
C06203=1059.866,301.777,399.487,173.335,34.995,156.535
C06204=1059.860,301.529,399.519,173.331,34.991,156.534
C06205=1059.853,301.282,399.551,173.328,34.987,156.533
C06206=1059.847,301.033,399.583,173.325,34.983,156.532
C06207=1059.840,300.786,399.616,173.321,34.978,156.532
C06208=1059.834,300.538,399.648,173.319,34.974,156.531
C06209=1059.828,300.290,399.679,173.316,34.971,156.530
C06210=1059.821,300.042,399.712,173.313,34.967,156.529
C06211=1059.815,299.794,399.744,173.309,34.963,156.528
C06212=1059.809,299.546,399.776,173.306,34.958,156.527
C06213=1059.804,299.299,399.808,173.304,34.954,156.527
C06214=1059.797,299.051,399.840,173.300,34.950,156.526
C06215=1059.791,298.803,399.872,173.297,34.946,156.525
C06216=1059.785,298.555,399.904,173.294,34.942,156.524
C06217=1059.779,298.307,399.936,173.290,34.938,156.523
C06218=1059.772,298.059,399.969,173.288,34.934,156.522
C06219=1059.766,297.812,400.000,173.285,34.930,156.522
C06220=1059.760,297.564,400.032,173.282,34.926,156.521
C06221=1059.754,297.316,400.065,173.278,34.922,156.520
C06222=1059.747,297.068,400.096,173.276,34.918,156.519
C06223=1059.741,296.820,400.128,173.273,34.914,156.518
C06224=1059.735,296.572,400.160,173.269,34.910,156.517
C06225=1059.729,296.325,400.192,173.266,34.906,156.517
C06226=1059.722,296.077,400.224,173.263,34.902,156.516
C06227=1059.716,295.829,400.256,173.261,34.898,156.515
C06228=1059.709,295.581,400.287,173.257,34.894,156.514
C06229=1059.704,295.333,400.319,173.254,34.890,156.513
C06230=1059.697,295.085,400.351,173.251,34.886,156.512
C06231=1059.691,294.838,400.382,173.248,34.882,156.512
C06232=1059.685,294.590,400.414,173.245,34.878,156.511
C06233=1059.678,294.342,400.445,173.242,34.874,156.510
C06234=1059.672,294.094,400.477,173.239,34.870,156.509
C06235=1059.665,293.846,400.509,173.236,34.866,156.508
C06236=1059.659,293.598,400.540,173.233,34.862,156.508
C06237=1059.653,293.350,400.572,173.230,34.859,156.507
C06238=1059.646,293.102,400.603,173.227,34.855,156.506
C06239=1059.640,292.854,400.635,173.224,34.850,156.505
C06240=1059.634,292.606,400.667,173.221,34.847,156.504
C06241=1059.628,292.359,400.698,173.218,34.843,156.504
C06242=1059.621,292.111,400.729,173.214,34.839,156.503
C06243=1059.615,291.863,400.761,173.212,34.835,156.502
C06244=1059.608,291.614,400.792,173.209,34.831,156.501
C06245=1059.602,291.378,400.822,173.206,34.827,156.500
C06246=1059.597,291.140,400.852,173.203,34.823,156.500
C06247=1059.590,290.903,400.882,173.200,34.820,156.499
C06248=1059.584,290.666,400.912,173.198,34.816,156.498
C06249=1059.579,290.429,400.943,173.195,34.813,156.497
C06250=1059.573,290.192,400.972,173.191,34.808,156.497
C06251=1059.566,289.954,401.002,173.189,34.805,156.496
C06252=1059.560,289.717,401.032,173.186,34.801,156.495
C06253=1059.554,289.469,401.064,173.184,34.797,156.494
C06254=1059.548,289.221,401.094,173.180,34.793,156.493
C06255=1059.542,288.973,401.125,173.177,34.789,156.493
C06256=1059.535,288.726,401.157,173.175,34.785,156.492
C06257=1059.529,288.477,401.189,173.172,34.782,156.491
C06258=1059.523,288.230,401.219,173.168,34.778,156.490
C06259=1059.516,287.982,401.251,173.165,34.774,156.490
C06260=1059.510,287.733,401.281,173.163,34.770,156.489
C06261=1059.504,287.486,401.312,173.160,34.766,156.488
C06262=1059.498,287.237,401.343,173.156,34.762,156.487
C06263=1059.491,286.989,401.375,173.154,34.759,156.486
C06264=1059.485,286.742,401.406,173.151,34.754,156.486
C06265=1059.478,286.494,401.436,173.148,34.751,156.485
C06266=1059.472,286.246,401.468,173.145,34.747,156.484
C06267=1059.466,285.998,401.498,173.142,34.743,156.483
C06268=1059.459,285.750,401.530,173.139,34.739,156.482
C06269=1059.453,285.502,401.560,173.137,34.735,156.482
C06270=1059.446,285.254,401.591,173.133,34.731,156.481
C06271=1059.440,285.006,401.622,173.130,34.728,156.480
C06272=1059.434,284.758,401.652,173.128,34.724,156.479
C06273=1059.427,284.510,401.684,173.125,34.720,156.479
C06274=1059.421,284.262,401.715,173.122,34.716,156.478
C06275=1059.415,284.014,401.746,173.119,34.712,156.477
C06276=1059.409,283.766,401.776,173.116,34.709,156.476
C06277=1059.403,283.518,401.807,173.114,34.705,156.475
C06278=1059.396,283.270,401.838,173.110,34.701,156.475
C06279=1059.390,283.022,401.868,173.107,34.697,156.474
C06280=1059.384,282.774,401.899,173.105,34.693,156.473
C06281=1059.377,282.526,401.931,173.102,34.689,156.472
C06282=1059.371,282.278,401.961,173.100,34.686,156.472
C06283=1059.365,282.030,401.992,173.096,34.681,156.471
C06284=1059.359,281.782,402.022,173.093,34.678,156.470
C06285=1059.352,281.534,402.053,173.091,34.674,156.469
C06286=1059.346,281.286,402.084,173.088,34.670,156.468
C06287=1059.340,281.037,402.115,173.085,34.666,156.468
C06288=1059.334,280.790,402.145,173.082,34.662,156.467
C06289=1059.327,280.542,402.176,173.079,34.658,156.466
C06290=1059.322,280.294,402.207,173.077,34.655,156.465
C06291=1059.316,280.046,402.237,173.073,34.650,156.465
C06292=1059.309,279.798,402.268,173.071,34.647,156.464
C06293=1059.304,279.550,402.298,173.068,34.643,156.463
C06294=1059.296,279.302,402.328,173.066,34.639,156.462
C06295=1059.291,279.054,402.359,173.062,34.636,156.462
C06296=1059.284,278.805,402.389,173.059,34.632,156.461
C06297=1059.278,278.557,402.420,173.057,34.628,156.460
C06298=1059.271,278.309,402.450,173.054,34.624,156.459
C06299=1059.265,278.061,402.480,173.052,34.620,156.458
C06300=1059.259,277.813,402.511,173.048,34.616,156.458
C06301=1059.253,277.581,402.540,173.046,34.613,156.457
C06302=1059.247,277.350,402.568,173.043,34.609,156.456
C06303=1059.242,277.118,402.596,173.041,34.606,156.456
C06304=1059.236,276.886,402.624,173.038,34.602,156.455
C06305=1059.230,276.654,402.653,173.035,34.599,156.454
C06306=1059.224,276.423,402.681,173.033,34.595,156.453
C06307=1059.218,276.191,402.710,173.030,34.591,156.453
C06308=1059.212,275.958,402.738,173.028,34.588,156.452
C06309=1059.206,275.711,402.767,173.025,34.584,156.451
C06310=1059.199,275.462,402.798,173.022,34.581,156.451
C06311=1059.194,275.215,402.829,173.020,34.576,156.450
C06312=1059.187,274.967,402.858,173.017,34.573,156.449
C06313=1059.181,274.718,402.888,173.014,34.569,156.448
C06314=1059.175,274.470,402.919,173.011,34.565,156.447
C06315=1059.169,274.223,402.948,173.008,34.562,156.447
C06316=1059.162,273.974,402.979,173.006,34.558,156.446
C06317=1059.156,273.726,403.009,173.003,34.554,156.445
C06318=1059.149,273.477,403.039,173.000,34.550,156.444
C06319=1059.144,273.230,403.069,172.997,34.547,156.444
C06320=1059.138,272.982,403.100,172.995,34.542,156.443
C06321=1059.131,272.734,403.129,172.992,34.539,156.442
C06322=1059.125,272.485,403.159,172.990,34.535,156.441
C06323=1059.119,272.238,403.189,172.986,34.531,156.441
C06324=1059.112,271.989,403.220,172.984,34.527,156.440
C06325=1059.106,271.741,403.249,172.981,34.524,156.439
C06326=1059.100,271.493,403.279,172.979,34.520,156.438
C06327=1059.094,271.245,403.308,172.976,34.516,156.438
C06328=1059.087,270.996,403.339,172.973,34.513,156.437
C06329=1059.081,270.749,403.369,172.970,34.509,156.436
C06330=1059.075,270.500,403.398,172.968,34.505,156.435
C06331=1059.068,270.252,403.428,172.965,34.501,156.435
C06332=1059.063,270.004,403.458,172.963,34.498,156.434
C06333=1059.056,269.756,403.488,172.960,34.493,156.433
C06334=1059.051,269.508,403.517,172.957,34.490,156.432
C06335=1059.043,269.260,403.548,172.955,34.486,156.432
C06336=1059.038,269.011,403.577,172.952,34.483,156.431
C06337=1059.031,268.764,403.607,172.949,34.478,156.430
C06338=1059.025,268.516,403.636,172.946,34.475,156.429
C06339=1059.019,268.267,403.667,172.944,34.471,156.429
C06340=1059.012,268.019,403.696,172.941,34.468,156.428
C06341=1059.006,267.771,403.726,172.939,34.463,156.427
C06342=1059.000,267.522,403.756,172.936,34.460,156.426
C06343=1058.994,267.274,403.785,172.933,34.456,156.426
C06344=1058.987,267.027,403.814,172.930,34.453,156.425
C06345=1058.982,266.778,403.844,172.928,34.448,156.424
C06346=1058.975,266.530,403.873,172.926,34.445,156.423
C06347=1058.968,266.282,403.903,172.923,34.441,156.423
C06348=1058.963,266.033,403.933,172.920,34.438,156.422
C06349=1058.956,265.785,403.962,172.917,34.433,156.421
C06350=1058.950,265.538,403.992,172.915,34.430,156.420
C06351=1058.944,265.289,404.021,172.912,34.426,156.420
C06352=1058.937,265.040,404.051,172.910,34.423,156.419
C06353=1058.931,264.792,404.080,172.907,34.419,156.418
C06354=1058.925,264.545,404.110,172.904,34.415,156.417
C06355=1058.919,264.296,404.139,172.902,34.411,156.417
C06356=1058.913,264.048,404.168,172.899,34.407,156.416
C06357=1058.907,263.818,404.196,172.897,34.404,156.415
C06358=1058.901,263.589,404.222,172.894,34.400,156.415
C06359=1058.896,263.359,404.250,172.892,34.397,156.414
C06360=1058.890,263.129,404.277,172.890,34.393,156.413
C06361=1058.885,262.899,404.304,172.887,34.390,156.413
C06362=1058.878,262.669,404.331,172.885,34.387,156.412
C06363=1058.872,262.439,404.358,172.883,34.383,156.411
C06364=1058.866,262.209,404.385,172.880,34.380,156.411
C06365=1058.859,261.961,404.414,172.877,34.376,156.410
C06366=1058.853,261.713,404.443,172.875,34.372,156.409
C06367=1058.847,261.465,404.473,172.872,34.369,156.408
C06368=1058.841,261.217,404.502,172.870,34.365,156.408
C06369=1058.834,260.968,404.531,172.867,34.361,156.407
C06370=1058.827,260.720,404.560,172.864,34.358,156.406
C06371=1058.821,260.472,404.589,172.862,34.354,156.406
C06372=1058.815,260.223,404.618,172.859,34.351,156.405
C06373=1058.809,259.975,404.647,172.857,34.347,156.404
C06374=1058.802,259.727,404.676,172.855,34.343,156.403
C06375=1058.797,259.478,404.704,172.851,34.339,156.403
C06376=1058.790,259.230,404.734,172.849,34.336,156.402
C06377=1058.783,258.981,404.763,172.847,34.332,156.401
C06378=1058.777,258.733,404.792,172.844,34.328,156.400
C06379=1058.771,258.485,404.821,172.842,34.325,156.400
C06380=1058.765,258.237,404.850,172.838,34.321,156.399
C06381=1058.758,257.989,404.878,172.836,34.318,156.398
C06382=1058.751,257.741,404.908,172.834,34.313,156.397
C06383=1058.746,257.492,404.936,172.831,34.310,156.397
C06384=1058.739,257.244,404.965,172.829,34.306,156.396
C06385=1058.733,256.996,404.994,172.827,34.303,156.395
C06386=1058.727,256.748,405.023,172.823,34.299,156.395
C06387=1058.721,256.500,405.052,172.821,34.295,156.394
C06388=1058.715,256.251,405.080,172.819,34.291,156.393
C06389=1058.708,256.003,405.109,172.816,34.287,156.392
C06390=1058.702,255.755,405.138,172.814,34.284,156.392
C06391=1058.696,255.507,405.167,172.812,34.280,156.391
C06392=1058.689,255.258,405.195,172.808,34.277,156.390
C06393=1058.683,255.010,405.224,172.806,34.273,156.390
C06394=1058.677,254.762,405.253,172.804,34.269,156.389
C06395=1058.671,254.513,405.282,172.801,34.265,156.388
C06396=1058.664,254.265,405.311,172.799,34.262,156.387
C06397=1058.658,254.017,405.340,172.797,34.258,156.387
C06398=1058.652,253.768,405.368,172.794,34.254,156.386
C06399=1058.646,253.520,405.397,172.791,34.250,156.385
C06400=1058.640,253.271,405.425,172.789,34.247,156.384
C06401=1058.633,253.023,405.454,172.787,34.243,156.384
C06402=1058.627,252.775,405.483,172.784,34.239,156.383
C06403=1058.621,252.527,405.511,172.781,34.235,156.382
C06404=1058.615,252.279,405.540,172.779,34.231,156.381
C06405=1058.609,252.030,405.568,172.777,34.228,156.381
C06406=1058.603,251.782,405.597,172.774,34.224,156.380
C06407=1058.597,251.534,405.626,172.772,34.221,156.379
C06408=1058.590,251.286,405.654,172.770,34.216,156.378
C06409=1058.584,251.037,405.682,172.766,34.213,156.378
C06410=1058.578,250.789,405.711,172.764,34.209,156.377
C06411=1058.572,250.540,405.740,172.762,34.206,156.376
C06412=1058.566,250.292,405.769,172.760,34.201,156.375
C06413=1058.560,250.062,405.795,172.758,34.198,156.375
C06414=1058.555,249.830,405.821,172.755,34.195,156.374
C06415=1058.549,249.599,405.848,172.753,34.191,156.374
C06416=1058.544,249.369,405.874,172.750,34.187,156.373
C06417=1058.537,249.138,405.901,172.748,34.184,156.372
C06418=1058.531,248.907,405.927,172.746,34.180,156.371
C06419=1058.526,248.675,405.953,172.744,34.177,156.371
C06420=1058.520,248.445,405.980,172.742,34.174,156.370
C06421=1058.514,248.196,406.008,172.740,34.170,156.369
C06422=1058.508,247.948,406.037,172.737,34.166,156.369
C06423=1058.503,247.700,406.065,172.734,34.162,156.368
C06424=1058.497,247.451,406.093,172.732,34.159,156.367
C06425=1058.490,247.204,406.122,172.730,34.154,156.366
C06426=1058.484,246.955,406.150,172.728,34.151,156.366
C06427=1058.479,246.707,406.178,172.725,34.147,156.365
C06428=1058.472,246.459,406.207,172.723,34.143,156.364
C06429=1058.466,246.210,406.235,172.720,34.139,156.363
C06430=1058.460,245.961,406.263,172.718,34.136,156.363
C06431=1058.454,245.713,406.291,172.716,34.132,156.362
C06432=1058.448,245.465,406.319,172.713,34.128,156.361
C06433=1058.441,245.217,406.348,172.711,34.124,156.360
C06434=1058.435,244.968,406.376,172.709,34.121,156.360
C06435=1058.429,244.720,406.404,172.706,34.117,156.359
C06436=1058.423,244.472,406.432,172.704,34.113,156.358
C06437=1058.417,244.223,406.460,172.701,34.110,156.358
C06438=1058.411,243.974,406.488,172.699,34.105,156.357
C06439=1058.404,243.727,406.516,172.697,34.102,156.356
C06440=1058.399,243.479,406.544,172.695,34.098,156.355
C06441=1058.392,243.230,406.572,172.693,34.095,156.355
C06442=1058.386,242.981,406.600,172.689,34.091,156.354
C06443=1058.379,242.733,406.628,172.687,34.087,156.353
C06444=1058.374,242.485,406.656,172.685,34.083,156.352
C06445=1058.367,242.236,406.684,172.683,34.079,156.352
C06446=1058.361,241.988,406.712,172.681,34.076,156.351
C06447=1058.355,241.740,406.739,172.679,34.072,156.350
C06448=1058.349,241.491,406.768,172.675,34.068,156.350
C06449=1058.343,241.243,406.796,172.673,34.064,156.349
C06450=1058.336,240.994,406.823,172.671,34.061,156.348
C06451=1058.331,240.746,406.851,172.669,34.057,156.347
C06452=1058.324,240.498,406.879,172.667,34.053,156.347
C06453=1058.317,240.249,406.907,172.664,34.050,156.346
C06454=1058.312,240.000,406.934,172.662,34.046,156.345
C06455=1058.305,239.752,406.962,172.659,34.042,156.344
C06456=1058.299,239.504,406.989,172.657,34.038,156.344
C06457=1058.293,239.255,407.018,172.655,34.035,156.343
C06458=1058.287,239.007,407.045,172.653,34.031,156.342
C06459=1058.280,238.759,407.073,172.651,34.027,156.342
C06460=1058.274,238.510,407.101,172.648,34.023,156.341
C06461=1058.268,238.262,407.128,172.646,34.020,156.340
C06462=1058.262,238.013,407.155,172.643,34.016,156.339
C06463=1058.255,237.765,407.183,172.641,34.012,156.339
C06464=1058.250,237.517,407.211,172.639,34.009,156.338
C06465=1058.243,237.268,407.238,172.637,34.005,156.337
C06466=1058.237,237.019,407.266,172.635,34.001,156.336
C06467=1058.230,236.772,407.293,172.632,33.997,156.336
C06468=1058.225,236.523,407.322,172.630,33.994,156.335
C06469=1058.218,236.289,407.346,172.628,33.990,156.334
C06470=1058.212,236.055,407.373,172.625,33.986,156.334
C06471=1058.207,235.821,407.398,172.623,33.983,156.333
C06472=1058.201,235.587,407.425,172.621,33.979,156.332
C06473=1058.195,235.353,407.450,172.619,33.976,156.332
C06474=1058.189,235.119,407.476,172.617,33.972,156.331
C06475=1058.184,234.885,407.502,172.615,33.969,156.330
C06476=1058.177,234.651,407.528,172.613,33.965,156.330
C06477=1058.172,234.403,407.555,172.611,33.961,156.329
C06478=1058.166,234.154,407.583,172.608,33.957,156.328
C06479=1058.160,233.907,407.611,172.606,33.954,156.327
C06480=1058.153,233.657,407.638,172.604,33.950,156.327
C06481=1058.147,233.409,407.665,172.602,33.946,156.326
C06482=1058.142,233.160,407.693,172.600,33.942,156.325
C06483=1058.135,232.912,407.720,172.598,33.939,156.324
C06484=1058.129,232.664,407.747,172.596,33.935,156.324
C06485=1058.122,232.415,407.775,172.593,33.931,156.323
C06486=1058.117,232.167,407.801,172.590,33.928,156.322
C06487=1058.110,231.918,407.829,172.588,33.923,156.322
C06488=1058.104,231.670,407.856,172.586,33.920,156.321
C06489=1058.098,231.422,407.883,172.584,33.916,156.320
C06490=1058.092,231.173,407.910,172.582,33.912,156.319
C06491=1058.085,230.925,407.938,172.580,33.908,156.319
C06492=1058.079,230.676,407.964,172.578,33.905,156.318
C06493=1058.073,230.428,407.992,172.575,33.901,156.317
C06494=1058.068,230.179,408.019,172.573,33.897,156.317
C06495=1058.061,229.930,408.046,172.571,33.893,156.316
C06496=1058.055,229.682,408.074,172.569,33.889,156.315
C06497=1058.049,229.433,408.101,172.567,33.886,156.314
C06498=1058.043,229.186,408.128,172.565,33.882,156.314
C06499=1058.036,228.937,408.155,172.563,33.878,156.313
C06500=1058.030,228.689,408.181,172.561,33.874,156.312
C06501=1058.023,228.439,408.208,172.558,33.871,156.311
C06502=1058.017,228.192,408.236,172.555,33.867,156.311
C06503=1058.011,227.943,408.263,172.553,33.863,156.310
C06504=1058.005,227.694,408.289,172.551,33.860,156.309
C06505=1057.998,227.446,408.317,172.549,33.855,156.308
C06506=1057.993,227.198,408.344,172.547,33.852,156.308
C06507=1057.986,226.949,408.370,172.545,33.848,156.307
C06508=1057.980,226.700,408.397,172.543,33.845,156.306
C06509=1057.973,226.452,408.424,172.541,33.840,156.306
C06510=1057.967,226.204,408.451,172.538,33.837,156.305
C06511=1057.961,225.955,408.478,172.536,33.833,156.304
C06512=1057.955,225.706,408.505,172.534,33.829,156.303
C06513=1057.949,225.458,408.531,172.532,33.826,156.303
C06514=1057.942,225.209,408.558,172.530,33.822,156.302
C06515=1057.936,224.961,408.585,172.528,33.818,156.301
C06516=1057.930,224.712,408.612,172.526,33.814,156.301
C06517=1057.924,224.464,408.639,172.524,33.810,156.300
C06518=1057.918,224.216,408.666,172.521,33.806,156.299
C06519=1057.911,223.967,408.692,172.519,33.803,156.298
C06520=1057.905,223.718,408.719,172.517,33.799,156.298
C06521=1057.900,223.470,408.745,172.515,33.795,156.297
C06522=1057.893,223.221,408.772,172.513,33.791,156.296
C06523=1057.888,222.973,408.799,172.511,33.788,156.295
C06524=1057.880,222.724,408.825,172.509,33.783,156.295
C06525=1057.875,222.486,408.851,172.507,33.780,156.294
C06526=1057.869,222.249,408.877,172.505,33.776,156.293
C06527=1057.863,222.011,408.902,172.503,33.772,156.293
C06528=1057.857,221.773,408.928,172.501,33.769,156.292
C06529=1057.851,221.536,408.953,172.499,33.765,156.291
C06530=1057.845,221.297,408.979,172.497,33.761,156.290
C06531=1057.840,221.059,409.004,172.495,33.758,156.290
C06532=1057.834,220.821,409.030,172.493,33.754,156.289
C06533=1057.827,220.573,409.056,172.491,33.751,156.288
C06534=1057.821,220.324,409.083,172.489,33.747,156.288
C06535=1057.815,220.075,409.109,172.487,33.743,156.287
C06536=1057.809,219.827,409.135,172.485,33.739,156.286
C06537=1057.803,219.578,409.162,172.482,33.735,156.285
C06538=1057.796,219.330,409.188,172.480,33.732,156.285
C06539=1057.790,219.082,409.215,172.478,33.727,156.284
C06540=1057.783,218.833,409.241,172.476,33.724,156.283
C06541=1057.777,218.585,409.268,172.474,33.720,156.283
C06542=1057.771,218.336,409.293,172.472,33.716,156.282
C06543=1057.765,218.087,409.320,172.470,33.712,156.281
C06544=1057.759,217.839,409.347,172.468,33.709,156.280
C06545=1057.753,217.591,409.373,172.466,33.705,156.280
C06546=1057.747,217.342,409.400,172.465,33.701,156.279
C06547=1057.740,217.093,409.425,172.462,33.697,156.278
C06548=1057.734,216.845,409.452,172.460,33.693,156.277
C06549=1057.728,216.596,409.478,172.458,33.689,156.277
C06550=1057.722,216.348,409.505,172.456,33.686,156.276
C06551=1057.715,216.099,409.530,172.454,33.682,156.275
C06552=1057.709,215.850,409.557,172.452,33.678,156.275
C06553=1057.703,215.602,409.583,172.450,33.674,156.274
C06554=1057.697,215.354,409.610,172.448,33.670,156.273
C06555=1057.690,215.105,409.635,172.446,33.666,156.272
C06556=1057.684,214.856,409.662,172.444,33.662,156.272
C06557=1057.678,214.608,409.688,172.441,33.659,156.271
C06558=1057.672,214.359,409.714,172.439,33.655,156.270
C06559=1057.666,214.111,409.740,172.438,33.651,156.269
C06560=1057.660,213.861,409.766,172.436,33.647,156.269
C06561=1057.653,213.613,409.792,172.434,33.643,156.268
C06562=1057.648,213.365,409.819,172.432,33.639,156.267
C06563=1057.641,213.116,409.844,172.430,33.635,156.266
C06564=1057.636,212.868,409.871,172.428,33.631,156.266
C06565=1057.629,212.619,409.896,172.426,33.628,156.265
C06566=1057.623,212.370,409.923,172.424,33.624,156.264
C06567=1057.617,212.122,409.949,172.422,33.620,156.263
C06568=1057.610,211.874,409.975,172.419,33.616,156.263
C06569=1057.605,211.625,410.001,172.418,33.612,156.262
C06570=1057.598,211.377,410.027,172.416,33.608,156.261
C06571=1057.592,211.129,410.053,172.414,33.604,156.260
C06572=1057.586,210.879,410.079,172.412,33.600,156.260
C06573=1057.579,210.631,410.105,172.410,33.597,156.259
C06574=1057.573,210.382,410.130,172.408,33.593,156.258
C06575=1057.568,210.133,410.156,172.406,33.589,156.257
C06576=1057.561,209.885,410.182,172.404,33.585,156.257
C06577=1057.555,209.636,410.208,172.403,33.581,156.256
C06578=1057.549,209.388,410.234,172.401,33.577,156.255
C06579=1057.542,209.139,410.260,172.398,33.573,156.254
C06580=1057.536,208.890,410.286,172.396,33.569,156.254
C06581=1057.530,208.655,410.311,172.394,33.566,156.253
C06582=1057.524,208.420,410.335,172.392,33.562,156.252
C06583=1057.518,208.184,410.359,172.391,33.559,156.252
C06584=1057.513,207.950,410.383,172.389,33.555,156.251
C06585=1057.507,207.715,410.408,172.387,33.551,156.250
C06586=1057.501,207.479,410.432,172.385,33.548,156.250
C06587=1057.495,207.244,410.456,172.384,33.544,156.249
C06588=1057.489,207.008,410.480,172.382,33.540,156.248
C06589=1057.464,205.958,410.586,172.188,33.452,156.236
C06590=1057.458,205.709,410.610,172.185,33.449,156.236
C06591=1057.452,205.460,410.635,172.183,33.445,156.235
C06592=1057.447,205.211,410.660,172.181,33.442,156.235
C06593=1057.440,204.963,410.684,172.178,33.439,156.234
C06594=1057.434,204.714,410.709,172.176,33.437,156.234
C06595=1057.428,204.466,410.734,172.174,33.433,156.233
C06596=1057.422,204.217,410.759,172.171,33.430,156.233
C06597=1057.417,203.969,410.784,172.169,33.427,156.232
C06598=1057.411,203.719,410.808,172.167,33.424,156.232
C06599=1057.405,203.470,410.833,172.165,33.422,156.231
C06600=1057.399,203.222,410.858,172.162,33.418,156.231
C06601=1057.393,202.973,410.882,172.160,33.415,156.230
C06602=1057.387,202.725,410.907,172.158,33.412,156.229
C06603=1057.381,202.476,410.932,172.155,33.409,156.229
C06604=1057.376,202.227,410.956,172.153,33.406,156.228
C06605=1057.370,201.979,410.981,172.151,33.403,156.228
C06606=1057.364,201.729,411.006,172.148,33.400,156.227
C06607=1057.358,201.481,411.029,172.146,33.397,156.227
C06608=1057.352,201.232,411.055,172.144,33.394,156.226
C06609=1057.346,200.984,411.078,172.142,33.391,156.226
C06610=1057.340,200.735,411.103,172.139,33.389,156.225
C06611=1057.333,200.486,411.127,172.136,33.386,156.225
C06612=1057.328,200.237,411.151,172.134,33.382,156.224
C06613=1057.321,199.989,411.177,172.131,33.380,156.224
C06614=1057.315,199.740,411.200,172.129,33.377,156.223
C06615=1057.310,199.491,411.225,172.127,33.374,156.223
C06616=1057.303,199.242,411.249,172.124,33.371,156.222
C06617=1057.298,198.993,411.273,172.122,33.368,156.222
C06618=1057.291,198.745,411.298,172.120,33.365,156.221
C06619=1057.285,198.496,411.322,172.118,33.362,156.221
C06620=1057.279,198.247,411.346,172.115,33.360,156.220
C06621=1057.273,197.999,411.370,172.113,33.356,156.220
C06622=1057.268,197.750,411.395,172.111,33.353,156.219
C06623=1057.261,197.501,411.419,172.109,33.351,156.219
C06624=1057.256,197.252,411.443,172.106,33.348,156.218
C06625=1057.250,197.004,411.467,172.104,33.345,156.218
C06626=1057.244,196.754,411.492,172.102,33.342,156.217
C06627=1057.237,196.507,411.516,172.100,33.339,156.217
C06628=1057.231,196.258,411.541,172.097,33.336,156.216
C06629=1057.225,196.009,411.564,172.095,33.333,156.216
C06630=1057.219,195.760,411.589,172.093,33.330,156.215
C06631=1057.213,195.512,411.613,172.091,33.327,156.214
C06632=1057.208,195.262,411.637,172.088,33.325,156.214
C06633=1057.201,195.014,411.661,172.086,33.322,156.214
C06634=1057.196,194.765,411.686,172.084,33.319,156.213
C06635=1057.190,194.517,411.709,172.082,33.316,156.213
C06636=1057.184,194.267,411.734,172.079,33.313,156.212
C06637=1057.178,194.019,411.757,172.077,33.310,156.212
C06638=1057.173,193.770,411.781,172.075,33.307,156.211
C06639=1057.166,193.521,411.805,172.073,33.304,156.211
C06640=1057.161,193.272,411.829,172.070,33.301,156.210
C06641=1057.154,193.023,411.853,172.068,33.299,156.210
C06642=1057.149,192.775,411.878,172.066,33.296,156.209
C06643=1057.142,192.526,411.902,172.064,33.293,156.209
C06644=1057.137,192.277,411.926,172.062,33.290,156.208
C06645=1057.131,192.029,411.950,172.059,33.287,156.208
C06646=1057.125,191.780,411.974,172.057,33.284,156.207
C06647=1057.119,191.531,411.997,172.055,33.282,156.207
C06648=1057.114,191.282,412.021,172.053,33.278,156.206
C06649=1057.107,191.033,412.045,172.051,33.275,156.205
C06650=1057.100,190.750,412.073,172.048,33.272,156.205
C06651=1057.094,190.465,412.100,172.046,33.269,156.204
C06652=1057.087,190.182,412.128,172.043,33.266,156.204
C06653=1057.081,189.898,412.155,172.041,33.263,156.203
C06654=1057.075,189.649,412.178,172.037,33.259,156.203
C06655=1057.069,189.400,412.203,172.035,33.257,156.202
C06656=1057.063,189.151,412.226,172.033,33.254,156.202
C06657=1057.058,188.903,412.250,172.031,33.251,156.201
C06658=1057.052,188.654,412.274,172.029,33.248,156.201
C06659=1057.046,188.404,412.298,172.027,33.246,156.200
C06660=1057.040,188.156,412.321,172.024,33.242,156.200
C06661=1057.035,187.908,412.346,172.022,33.240,156.199
C06662=1057.028,187.659,412.370,172.020,33.237,156.199
C06663=1057.022,187.410,412.393,172.018,33.234,156.198
C06664=1057.017,187.161,412.417,172.016,33.231,156.198
C06665=1057.011,186.913,412.441,172.014,33.228,156.197
C06666=1057.006,186.663,412.465,172.012,33.225,156.197
C06667=1057.000,186.415,412.488,172.009,33.223,156.196
C06668=1056.995,186.165,412.512,172.007,33.219,156.196
C06669=1056.988,185.917,412.535,172.005,33.217,156.195
C06670=1056.982,185.668,412.559,172.003,33.214,156.195
C06671=1056.977,185.419,412.583,172.001,33.211,156.194
C06672=1056.971,185.171,412.607,171.999,33.208,156.194
C06673=1056.966,184.922,412.630,171.997,33.206,156.193
C06674=1056.960,184.673,412.654,171.994,33.202,156.193
C06675=1056.953,184.424,412.677,171.992,33.200,156.192
C06676=1056.948,184.175,412.701,171.990,33.197,156.192
C06677=1056.942,183.927,412.724,171.988,33.194,156.191
C06678=1056.935,183.678,412.748,171.986,33.192,156.191
C06679=1056.929,183.429,412.771,171.984,33.189,156.190
C06680=1056.923,183.180,412.794,171.982,33.186,156.190
C06681=1056.917,182.931,412.818,171.979,33.183,156.189
C06682=1056.911,182.682,412.841,171.977,33.181,156.189
C06683=1056.905,182.434,412.864,171.975,33.178,156.189
C06684=1056.899,182.185,412.887,171.973,33.176,156.188
C06685=1056.893,181.936,412.911,171.971,33.172,156.188
C06686=1056.887,181.687,412.934,171.969,33.170,156.187
C06687=1056.881,181.438,412.957,171.967,33.167,156.187
C06688=1056.875,181.189,412.981,171.964,33.165,156.186
C06689=1056.869,180.940,413.004,171.962,33.162,156.186
C06690=1056.863,180.691,413.026,171.960,33.160,156.185
C06691=1056.856,180.443,413.050,171.958,33.156,156.185
C06692=1056.850,180.194,413.073,171.956,33.154,156.184
C06693=1056.844,179.945,413.096,171.954,33.151,156.184
C06694=1056.838,179.696,413.120,171.952,33.149,156.183
C06695=1056.833,179.448,413.143,171.950,33.146,156.183
C06696=1056.827,179.199,413.166,171.947,33.143,156.182
C06697=1056.821,178.949,413.189,171.945,33.140,156.182
C06698=1056.815,178.701,413.213,171.943,33.138,156.182
C06699=1056.808,178.452,413.235,171.941,33.135,156.181
C06700=1056.802,178.203,413.258,171.939,33.133,156.181
C06701=1056.797,177.954,413.281,171.937,33.130,156.180
C06702=1056.790,177.705,413.304,171.935,33.127,156.180
C06703=1056.784,177.456,413.328,171.933,33.124,156.179
C06704=1056.779,177.208,413.351,171.931,33.122,156.179
C06705=1056.773,176.959,413.374,171.929,33.119,156.178
C06706=1056.767,176.710,413.397,171.926,33.117,156.178
C06707=1056.761,176.461,413.419,171.924,33.114,156.177
C06708=1056.754,176.212,413.443,171.922,33.111,156.177
C06709=1056.748,175.963,413.466,171.920,33.108,156.177
C06710=1056.742,175.714,413.489,171.918,33.106,156.176
C06711=1056.737,175.466,413.512,171.916,33.103,156.176
C06712=1056.731,175.217,413.535,171.914,33.100,156.175
C06713=1056.725,174.968,413.558,171.912,33.098,156.175
C06714=1056.718,174.684,413.584,171.909,33.094,156.174
C06715=1056.711,174.399,413.610,171.907,33.092,156.174
C06716=1056.705,174.115,413.636,171.905,33.089,156.173
C06717=1056.698,173.831,413.663,171.902,33.085,156.173
C06718=1056.692,173.582,413.686,171.900,33.083,156.172
C06719=1056.686,173.333,413.709,171.898,33.080,156.172
C06720=1056.680,173.085,413.731,171.896,33.078,156.171
C06721=1056.674,172.835,413.754,171.894,33.075,156.171
C06722=1056.668,172.586,413.777,171.892,33.072,156.170
C06723=1056.662,172.337,413.800,171.890,33.069,156.170
C06724=1056.656,172.088,413.823,171.888,33.067,156.169
C06725=1056.650,171.840,413.846,171.886,33.064,156.169
C06726=1056.644,171.591,413.869,171.884,33.062,156.169
C06727=1056.638,171.342,413.891,171.882,33.059,156.168
C06728=1056.633,171.093,413.914,171.880,33.056,156.168
C06729=1056.627,170.844,413.937,171.878,33.053,156.167
C06730=1056.621,170.595,413.960,171.876,33.051,156.167
C06731=1056.615,170.347,413.983,171.874,33.048,156.166
C06732=1056.609,170.097,414.005,171.872,33.046,156.166
C06733=1056.604,169.848,414.028,171.870,33.043,156.165
C06734=1056.598,169.599,414.051,171.868,33.040,156.165
C06735=1056.592,169.350,414.074,171.866,33.037,156.164
C06736=1056.586,169.102,414.096,171.864,33.035,156.164
C06737=1056.580,168.853,414.119,171.862,33.032,156.164
C06738=1056.574,168.604,414.142,171.860,33.029,156.163
C06739=1056.569,168.355,414.165,171.858,33.027,156.163
C06740=1056.562,168.106,414.187,171.856,33.024,156.162
C06741=1056.557,167.857,414.209,171.854,33.021,156.162
C06742=1056.551,167.608,414.232,171.852,33.019,156.161
C06743=1056.545,167.359,414.255,171.850,33.016,156.161
C06744=1056.539,167.111,414.277,171.848,33.013,156.160
C06745=1056.534,166.862,414.300,171.846,33.011,156.160
C06746=1056.528,166.613,414.323,171.844,33.008,156.159
C06747=1056.522,166.364,414.345,171.842,33.005,156.159
C06748=1056.517,166.115,414.368,171.840,33.003,156.158
C06749=1056.511,165.866,414.390,171.838,33.000,156.158
C06750=1056.505,165.617,414.413,171.836,32.997,156.158
C06751=1056.499,165.368,414.436,171.834,32.995,156.157
C06752=1056.493,165.119,414.459,171.832,32.992,156.157
C06753=1056.487,164.870,414.481,171.830,32.989,156.156
C06754=1056.482,164.622,414.503,171.828,32.987,156.156
C06755=1056.476,164.373,414.526,171.826,32.984,156.155
C06756=1056.471,164.123,414.548,171.824,32.981,156.155
C06757=1056.464,163.875,414.571,171.822,32.979,156.154
C06758=1056.459,163.626,414.594,171.820,32.976,156.154
C06759=1056.453,163.376,414.616,171.818,32.973,156.153
C06760=1056.447,163.128,414.638,171.816,32.971,156.153
C06761=1056.442,162.880,414.661,171.814,32.968,156.152
C06762=1056.436,162.630,414.683,171.812,32.965,156.152
C06763=1056.431,162.381,414.706,171.810,32.963,156.152
C06764=1056.424,162.132,414.728,171.808,32.960,156.151
C06765=1056.419,161.883,414.751,171.806,32.957,156.151
C06766=1056.413,161.635,414.773,171.804,32.955,156.150
C06767=1056.407,161.386,414.795,171.802,32.952,156.150
C06768=1056.402,161.137,414.818,171.800,32.949,156.149
C06769=1056.396,160.887,414.840,171.798,32.946,156.149
C06770=1056.390,160.639,414.862,171.796,32.944,156.148
C06771=1056.384,160.389,414.884,171.795,32.941,156.148
C06772=1056.378,160.141,414.907,171.793,32.939,156.148
C06773=1056.372,159.892,414.928,171.792,32.936,156.147
C06774=1056.367,159.643,414.951,171.790,32.934,156.147
C06775=1056.360,159.394,414.973,171.788,32.931,156.146
C06776=1056.354,159.145,414.995,171.786,32.929,156.146
C06777=1056.348,158.896,415.017,171.784,32.926,156.145
C06778=1056.342,158.611,415.043,171.781,32.923,156.145
C06779=1056.335,158.326,415.068,171.779,32.920,156.144
C06780=1056.327,158.042,415.093,171.777,32.918,156.144
C06781=1056.321,157.757,415.118,171.775,32.914,156.143
C06782=1056.316,157.508,415.140,171.773,32.912,156.143
C06783=1056.310,157.260,415.162,171.771,32.909,156.143
C06784=1056.303,157.011,415.184,171.769,32.907,156.142
C06785=1056.298,156.762,415.207,171.767,32.904,156.142
C06786=1056.291,156.512,415.228,171.765,32.901,156.141
C06787=1056.286,156.264,415.250,171.763,32.899,156.141
C06788=1056.280,156.015,415.273,171.761,32.896,156.140
C06789=1056.274,155.766,415.294,171.759,32.894,156.140
C06790=1056.268,155.517,415.316,171.757,32.891,156.140
C06791=1056.262,155.267,415.338,171.755,32.889,156.139
C06792=1056.257,155.019,415.360,171.753,32.886,156.139
C06793=1056.250,154.770,415.382,171.752,32.884,156.138
C06794=1056.244,154.521,415.403,171.750,32.881,156.138
C06795=1056.239,154.271,415.426,171.748,32.879,156.137
C06796=1056.232,154.023,415.448,171.746,32.876,156.137
C06797=1056.227,153.774,415.469,171.744,32.874,156.137
C06798=1056.221,153.525,415.491,171.742,32.871,156.136
C06799=1056.214,153.276,415.512,171.740,32.869,156.136
C06800=1056.209,153.027,415.535,171.738,32.866,156.135
C06801=1056.203,152.778,415.557,171.736,32.863,156.135
C06802=1056.197,152.529,415.578,171.734,32.861,156.134
C06803=1056.191,152.280,415.600,171.732,32.858,156.134
C06804=1056.185,152.031,415.622,171.730,32.856,156.134
C06805=1056.180,151.782,415.643,171.729,32.853,156.133
C06806=1056.173,151.533,415.666,171.727,32.851,156.133
C06807=1056.167,151.284,415.687,171.725,32.848,156.132
C06808=1056.162,151.036,415.709,171.723,32.845,156.132
C06809=1056.155,150.786,415.730,171.721,32.843,156.132
C06810=1056.149,150.537,415.752,171.719,32.841,156.131
C06811=1056.144,150.288,415.774,171.717,32.838,156.131
C06812=1056.138,150.039,415.796,171.715,32.836,156.130
C06813=1056.132,149.790,415.817,171.713,32.833,156.130
C06814=1056.126,149.541,415.839,171.711,32.831,156.129
C06815=1056.120,149.292,415.860,171.710,32.828,156.129
C06816=1056.114,149.043,415.882,171.708,32.825,156.129
C06817=1056.108,148.794,415.903,171.706,32.823,156.128
C06818=1056.103,148.545,415.925,171.704,32.820,156.128
C06819=1056.096,148.296,415.946,171.702,32.818,156.127
C06820=1056.091,148.047,415.968,171.700,32.816,156.127
C06821=1056.085,147.798,415.990,171.699,32.813,156.126
C06822=1056.079,147.549,416.011,171.697,32.811,156.126
C06823=1056.073,147.300,416.033,171.695,32.808,156.126
C06824=1056.067,147.051,416.055,171.694,32.805,156.125
C06825=1056.061,146.802,416.076,171.692,32.803,156.125
C06826=1056.055,146.553,416.098,171.690,32.800,156.124
C06827=1056.048,146.304,416.119,171.688,32.798,156.124
C06828=1056.043,146.055,416.140,171.686,32.796,156.124
C06829=1056.037,145.806,416.161,171.684,32.793,156.123
C06830=1056.030,145.557,416.183,171.682,32.791,156.123
C06831=1056.025,145.309,416.204,171.680,32.788,156.122
C06832=1056.019,145.059,416.226,171.679,32.786,156.122
C06833=1056.013,144.810,416.248,171.677,32.783,156.122
C06834=1056.007,144.561,416.268,171.675,32.781,156.121
C06835=1056.001,144.312,416.290,171.673,32.778,156.121
C06836=1055.996,144.063,416.311,171.671,32.776,156.120
C06837=1055.989,143.814,416.333,171.669,32.773,156.120
C06838=1055.983,143.565,416.354,171.667,32.771,156.119
C06839=1055.978,143.316,416.376,171.665,32.769,156.119
C06840=1055.971,143.067,416.396,171.664,32.766,156.119
C06841=1055.965,142.818,416.417,171.662,32.763,156.118
C06842=1055.959,142.533,416.442,171.660,32.761,156.118
C06843=1055.952,142.248,416.467,171.658,32.758,156.117
C06844=1055.945,141.963,416.491,171.655,32.755,156.117
C06845=1055.938,141.678,416.515,171.653,32.752,156.116
C06846=1055.932,141.430,416.536,171.651,32.750,156.116
C06847=1055.927,141.180,416.557,171.650,32.747,156.115
C06848=1055.921,140.931,416.579,171.648,32.745,156.115
C06849=1055.915,140.682,416.600,171.646,32.742,156.115
C06850=1055.909,140.433,416.622,171.644,32.739,156.114
C06851=1055.903,140.184,416.642,171.642,32.737,156.114
C06852=1055.897,139.935,416.664,171.640,32.734,156.113
C06853=1055.891,139.686,416.685,171.639,32.732,156.113
C06854=1055.885,139.436,416.706,171.637,32.730,156.113
C06855=1055.880,139.188,416.727,171.636,32.727,156.112
C06856=1055.873,138.939,416.748,171.634,32.725,156.112
C06857=1055.867,138.689,416.769,171.632,32.722,156.111
C06858=1055.861,138.441,416.790,171.630,32.720,156.111
C06859=1055.855,138.191,416.811,171.629,32.718,156.111
C06860=1055.849,137.943,416.832,171.627,32.715,156.110
C06861=1055.843,137.693,416.853,171.625,32.712,156.110
C06862=1055.838,137.444,416.874,171.623,32.710,156.109
C06863=1055.832,137.195,416.896,171.621,32.708,156.109
C06864=1055.826,136.946,416.916,171.619,32.705,156.108
C06865=1055.819,136.697,416.937,171.618,32.703,156.108
C06866=1055.814,136.449,416.958,171.616,32.700,156.108
C06867=1055.807,136.199,416.979,171.614,32.698,156.107
C06868=1055.802,135.951,417.000,171.612,32.695,156.107
C06869=1055.796,135.701,417.021,171.610,32.693,156.106
C06870=1055.789,135.453,417.042,171.608,32.690,156.106
C06871=1055.784,135.203,417.063,171.607,32.688,156.106
C06872=1055.778,134.954,417.084,171.605,32.686,156.105
C06873=1055.771,134.705,417.104,171.603,32.683,156.105
C06874=1055.766,134.456,417.125,171.601,32.681,156.104
C06875=1055.760,134.206,417.146,171.599,32.679,156.104
C06876=1055.754,133.958,417.167,171.598,32.676,156.104
C06877=1055.748,133.708,417.188,171.596,32.673,156.103
C06878=1055.742,133.460,417.208,171.594,32.671,156.103
C06879=1055.736,133.210,417.230,171.592,32.668,156.102
C06880=1055.730,132.961,417.250,171.590,32.666,156.102
C06881=1055.724,132.712,417.271,171.588,32.664,156.102
C06882=1055.718,132.463,417.292,171.587,32.661,156.101
C06883=1055.713,132.215,417.313,171.586,32.659,156.101
C06884=1055.706,131.965,417.333,171.584,32.657,156.100
C06885=1055.701,131.716,417.354,171.582,32.654,156.100
C06886=1055.694,131.467,417.375,171.580,32.651,156.100
C06887=1055.689,131.218,417.395,171.579,32.649,156.099
C06888=1055.682,130.969,417.416,171.577,32.647,156.099
C06889=1055.676,130.720,417.436,171.575,32.644,156.098
C06890=1055.670,130.471,417.457,171.573,32.642,156.098
C06891=1055.664,130.222,417.477,171.571,32.640,156.098
C06892=1055.658,129.973,417.499,171.570,32.637,156.097
C06893=1055.652,129.724,417.519,171.568,32.635,156.097
C06894=1055.645,129.474,417.539,171.566,32.632,156.096
C06895=1055.640,129.225,417.560,171.564,32.630,156.096
C06896=1055.633,128.976,417.581,171.562,32.628,156.096
C06897=1055.627,128.727,417.601,171.561,32.625,156.095
C06898=1055.622,128.478,417.621,171.559,32.623,156.095
C06899=1055.615,128.229,417.642,171.557,32.621,156.095
C06900=1055.609,127.981,417.662,171.555,32.618,156.094
C06901=1055.603,127.731,417.683,171.553,32.616,156.094
C06902=1055.597,127.482,417.703,171.552,32.614,156.093
C06903=1055.591,127.232,417.724,171.550,32.611,156.093
C06904=1055.585,126.983,417.744,171.548,32.608,156.093
C06905=1055.579,126.735,417.765,171.546,32.606,156.092
C06906=1055.572,126.450,417.788,171.544,32.604,156.092
C06907=1055.565,126.164,417.811,171.542,32.601,156.091
C06908=1055.559,125.879,417.835,171.541,32.598,156.091
C06909=1055.551,125.594,417.858,171.539,32.595,156.090
C06910=1055.546,125.345,417.878,171.537,32.593,156.090
C06911=1055.539,125.096,417.899,171.536,32.591,156.090
C06912=1055.533,124.847,417.919,171.534,32.588,156.089
C06913=1055.528,124.598,417.940,171.532,32.586,156.089
C06914=1055.521,124.348,417.960,171.530,32.584,156.089
C06915=1055.515,124.100,417.980,171.528,32.581,156.088
C06916=1055.509,123.850,418.001,171.527,32.579,156.088
C06917=1055.503,123.601,418.021,171.525,32.576,156.087
C06918=1055.497,123.352,418.041,171.523,32.574,156.087
C06919=1055.491,123.102,418.062,171.521,32.571,156.086
C06920=1055.485,122.854,418.082,171.520,32.569,156.086
C06921=1055.479,122.605,418.102,171.518,32.567,156.086
C06922=1055.473,122.355,418.122,171.516,32.564,156.085
C06923=1055.468,122.106,418.143,171.514,32.562,156.085
C06924=1055.462,121.857,418.163,171.513,32.560,156.085
C06925=1055.456,121.608,418.183,171.511,32.557,156.084
C06926=1055.450,121.359,418.204,171.509,32.554,156.084
C06927=1055.444,121.110,418.223,171.507,32.552,156.083
C06928=1055.438,120.861,418.243,171.506,32.550,156.083
C06929=1055.431,120.611,418.264,171.504,32.547,156.083
C06930=1055.426,120.362,418.284,171.503,32.545,156.082
C06931=1055.420,120.114,418.304,171.501,32.543,156.082
C06932=1055.414,119.865,418.324,171.500,32.540,156.081
C06933=1055.408,119.615,418.345,171.498,32.538,156.081
C06934=1055.402,119.366,418.365,171.496,32.536,156.081
C06935=1055.396,119.117,418.385,171.494,32.533,156.080
C06936=1055.390,118.868,418.405,171.493,32.530,156.080
C06937=1055.384,118.619,418.426,171.491,32.528,156.079
C06938=1055.378,118.370,418.446,171.489,32.526,156.079
C06939=1055.372,118.121,418.466,171.487,32.523,156.079
C06940=1055.366,117.872,418.486,171.486,32.521,156.078
C06941=1055.360,117.622,418.507,171.484,32.519,156.078
C06942=1055.355,117.373,418.526,171.482,32.516,156.077
C06943=1055.349,117.124,418.546,171.480,32.513,156.077
C06944=1055.343,116.875,418.566,171.479,32.511,156.077
C06945=1055.337,116.626,418.586,171.477,32.509,156.076
C06946=1055.331,116.377,418.607,171.475,32.506,156.076
C06947=1055.325,116.128,418.627,171.474,32.504,156.075
C06948=1055.319,115.878,418.646,171.472,32.501,156.075
C06949=1055.314,115.629,418.667,171.470,32.499,156.075
C06950=1055.308,115.381,418.687,171.468,32.496,156.074
C06951=1055.302,115.132,418.706,171.468,32.494,156.074
C06952=1055.295,114.882,418.727,171.466,32.491,156.073
C06953=1055.290,114.632,418.747,171.464,32.489,156.073
C06954=1055.284,114.384,418.767,171.462,32.487,156.073
C06955=1055.278,114.135,418.787,171.461,32.484,156.072
C06956=1055.272,113.886,418.807,171.459,32.482,156.072
C06957=1055.266,113.636,418.826,171.457,32.480,156.071
C06958=1055.260,113.387,418.846,171.456,32.477,156.071
C06959=1055.254,113.138,418.866,171.454,32.475,156.071
C06960=1055.248,112.889,418.886,171.452,32.472,156.070
C06961=1055.242,112.640,418.905,171.450,32.470,156.070
C06962=1055.236,112.391,418.925,171.449,32.468,156.070
C06963=1055.230,112.142,418.946,171.447,32.465,156.069
C06964=1055.224,111.892,418.965,171.445,32.463,156.069
C06965=1055.218,111.643,418.985,171.443,32.461,156.068
C06966=1055.212,111.395,419.005,171.442,32.458,156.068
C06967=1055.206,111.145,419.024,171.440,32.456,156.068
C06968=1055.200,110.896,419.044,171.438,32.453,156.067
C06969=1055.194,110.646,419.063,171.437,32.451,156.067
C06970=1055.187,110.362,419.086,171.435,32.448,156.066
C06971=1055.180,110.076,419.109,171.434,32.446,156.066
C06972=1055.173,109.791,419.131,171.432,32.443,156.065
C06973=1055.167,109.506,419.153,171.430,32.440,156.065
C06974=1055.160,109.256,419.173,171.428,32.438,156.065
C06975=1055.154,109.007,419.193,171.426,32.436,156.064
C06976=1055.148,108.758,419.213,171.424,32.433,156.064
C06977=1055.142,108.509,419.231,171.423,32.431,156.064
C06978=1055.136,108.260,419.251,171.421,32.429,156.063
C06979=1055.130,108.011,419.271,171.419,32.426,156.063
C06980=1055.124,107.762,419.290,171.418,32.424,156.062
C06981=1055.118,107.512,419.311,171.416,32.422,156.062
C06982=1055.112,107.263,419.330,171.414,32.419,156.062
C06983=1055.106,107.014,419.349,171.412,32.417,156.061
C06984=1055.100,106.765,419.369,171.411,32.415,156.061
C06985=1055.094,106.516,419.388,171.409,32.412,156.061
C06986=1055.088,106.267,419.408,171.407,32.410,156.060
C06987=1055.082,106.017,419.427,171.406,32.408,156.060
C06988=1055.076,105.769,419.447,171.405,32.405,156.059
C06989=1055.070,105.519,419.466,171.403,32.403,156.059
C06990=1055.063,105.270,419.486,171.402,32.401,156.059
C06991=1055.057,105.020,419.505,171.400,32.398,156.058
C06992=1055.052,104.771,419.524,171.398,32.396,156.058
C06993=1055.046,104.522,419.544,171.396,32.393,156.057
C06994=1055.039,104.273,419.563,171.395,32.391,156.057
C06995=1055.033,104.024,419.583,171.393,32.389,156.057
C06996=1055.028,103.775,419.602,171.391,32.386,156.056
C06997=1055.022,103.525,419.622,171.390,32.384,156.056
C06998=1055.016,103.277,419.641,171.388,32.382,156.056
C06999=1055.010,103.027,419.660,171.386,32.379,156.055
C07000=1055.004,102.778,419.679,171.385,32.377,156.055
C07001=1054.998,102.529,419.699,171.383,32.374,156.054
C07002=1054.992,102.280,419.719,171.381,32.372,156.054
C07003=1054.986,102.031,419.737,171.379,32.370,156.054
C07004=1054.980,101.782,419.757,171.378,32.367,156.053
C07005=1054.974,101.532,419.776,171.377,32.365,156.053
C07006=1054.968,101.283,419.796,171.375,32.363,156.052
C07007=1054.962,101.034,419.816,171.374,32.360,156.052
C07008=1054.956,100.785,419.834,171.372,32.358,156.052
C07009=1054.950,100.536,419.854,171.370,32.355,156.051
C07010=1054.945,100.286,419.873,171.369,32.354,156.051
C07011=1054.938,100.038,419.892,171.367,32.351,156.051
C07012=1054.932,99.788,419.911,171.365,32.349,156.050
C07013=1054.925,99.538,419.930,171.363,32.346,156.050
C07014=1054.920,99.289,419.950,171.362,32.344,156.050
C07015=1054.913,99.040,419.968,171.360,32.342,156.049
C07016=1054.907,98.791,419.988,171.358,32.340,156.049
C07017=1054.901,98.542,420.007,171.357,32.337,156.048
C07018=1054.895,98.293,420.026,171.355,32.334,156.048
C07019=1054.889,98.043,420.045,171.353,32.332,156.048
C07020=1054.883,97.794,420.064,171.352,32.330,156.047
C07021=1054.877,97.545,420.084,171.350,32.328,156.047
C07022=1054.870,97.296,420.103,171.349,32.325,156.046
C07023=1054.865,97.047,420.122,171.348,32.323,156.046
C07024=1054.858,96.797,420.141,171.346,32.321,156.046
C07025=1054.853,96.548,420.160,171.344,32.319,156.045
C07026=1054.846,96.299,420.178,171.342,32.316,156.045
C07027=1054.841,96.049,420.198,171.341,32.314,156.045
C07028=1054.834,95.800,420.216,171.339,32.311,156.044
C07029=1054.828,95.551,420.236,171.337,32.309,156.044
C07030=1054.822,95.303,420.255,171.336,32.307,156.044
C07031=1054.817,95.054,420.274,171.334,32.304,156.043
C07032=1054.810,94.805,420.292,171.332,32.302,156.043
C07033=1054.804,94.555,420.312,171.331,32.300,156.042
C07034=1054.798,94.270,420.333,171.329,32.297,156.042
C07035=1054.791,93.985,420.355,171.327,32.294,156.042
C07036=1054.783,93.699,420.377,171.325,32.292,156.041
C07037=1054.776,93.414,420.398,171.324,32.289,156.041
C07038=1054.771,93.164,420.417,171.322,32.287,156.040
C07039=1054.765,92.916,420.435,171.321,32.285,156.040
C07040=1054.759,92.666,420.455,171.319,32.282,156.040
C07041=1054.753,92.417,420.473,171.317,32.280,156.039
C07042=1054.747,92.168,420.493,171.316,32.277,156.039
C07043=1054.741,91.919,420.511,171.314,32.275,156.038
C07044=1054.735,91.669,420.530,171.312,32.273,156.038
C07045=1054.729,91.420,420.549,171.311,32.270,156.038
C07046=1054.723,91.171,420.568,171.309,32.268,156.037
C07047=1054.716,90.921,420.587,171.307,32.266,156.037
C07048=1054.711,90.672,420.606,171.306,32.264,156.037
C07049=1054.705,90.424,420.625,171.304,32.261,156.036
C07050=1054.698,90.175,420.643,171.302,32.259,156.036
C07051=1054.693,89.925,420.662,171.301,32.256,156.035
C07052=1054.686,89.676,420.681,171.300,32.254,156.035
C07053=1054.680,89.426,420.699,171.298,32.252,156.035
C07054=1054.674,89.177,420.718,171.297,32.250,156.034
C07055=1054.668,88.928,420.737,171.295,32.247,156.034
C07056=1054.662,88.679,420.756,171.293,32.245,156.034
C07057=1054.655,88.429,420.774,171.291,32.242,156.033
C07058=1054.649,88.180,420.793,171.290,32.241,156.033
C07059=1054.643,87.930,420.811,171.288,32.239,156.033
C07060=1054.638,87.682,420.830,171.286,32.236,156.032
C07061=1054.631,87.433,420.848,171.285,32.234,156.032
C07062=1054.625,87.184,420.867,171.283,32.231,156.031
C07063=1054.619,86.934,420.886,171.281,32.229,156.031
C07064=1054.613,86.684,420.904,171.280,32.227,156.031
C07065=1054.607,86.435,420.923,171.278,32.225,156.030
C07066=1054.600,86.186,420.941,171.276,32.222,156.030
C07067=1054.594,85.938,420.960,171.276,32.220,156.030
C07068=1054.589,85.688,420.978,171.274,32.217,156.029
C07069=1054.583,85.439,420.997,171.272,32.215,156.029
C07070=1054.576,85.189,421.016,171.271,32.213,156.029
C07071=1054.570,84.940,421.034,171.269,32.211,156.028
C07072=1054.564,84.691,421.052,171.267,32.208,156.028
C07073=1054.558,84.442,421.071,171.266,32.206,156.027
C07074=1054.552,84.193,421.090,171.264,32.204,156.027
C07075=1054.546,83.943,421.108,171.262,32.202,156.027
C07076=1054.539,83.694,421.126,171.261,32.199,156.026
C07077=1054.533,83.445,421.145,171.259,32.197,156.026
C07078=1054.528,83.195,421.163,171.257,32.194,156.026
C07079=1054.522,82.946,421.182,171.256,32.192,156.025
C07080=1054.515,82.697,421.200,171.254,32.190,156.025
C07081=1054.509,82.447,421.218,171.253,32.188,156.025
C07082=1054.503,82.198,421.237,171.252,32.185,156.024
C07083=1054.498,81.950,421.256,171.250,32.183,156.024
C07084=1054.492,81.700,421.274,171.248,32.181,156.023
C07085=1054.485,81.451,421.292,171.247,32.179,156.023
C07086=1054.479,81.201,421.310,171.245,32.176,156.023
C07087=1054.473,80.953,421.329,171.243,32.174,156.022
C07088=1054.468,80.703,421.348,171.242,32.171,156.022
C07089=1054.461,80.453,421.366,171.240,32.169,156.022
C07090=1054.455,80.204,421.384,171.238,32.167,156.021
C07091=1054.450,79.955,421.402,171.237,32.165,156.021
C07092=1054.443,79.706,421.421,171.235,32.162,156.020
C07093=1054.437,79.457,421.439,171.233,32.159,156.020
C07094=1054.432,79.208,421.457,171.232,32.158,156.020
C07095=1054.425,78.958,421.476,171.231,32.155,156.019
C07096=1054.419,78.709,421.494,171.229,32.153,156.019
C07097=1054.413,78.460,421.513,171.228,32.150,156.019
C07098=1054.406,78.174,421.533,171.226,32.148,156.018
C07099=1054.400,77.889,421.554,171.224,32.146,156.018
C07100=1054.392,77.604,421.575,171.222,32.143,156.017
C07101=1054.385,77.319,421.596,171.220,32.140,156.017
C07102=1054.379,77.069,421.614,171.219,32.138,156.017
C07103=1054.373,76.820,421.632,171.217,32.136,156.016
C07104=1054.367,76.571,421.650,171.215,32.133,156.016
C07105=1054.361,76.321,421.668,171.214,32.131,156.016
C07106=1054.355,76.072,421.686,171.212,32.129,156.015
C07107=1054.348,75.822,421.704,171.211,32.126,156.015
C07108=1054.343,75.574,421.723,171.210,32.125,156.015
C07109=1054.337,75.324,421.740,171.208,32.122,156.014
C07110=1054.330,75.074,421.758,171.206,32.120,156.014
C07111=1054.325,74.826,421.777,171.205,32.117,156.013
C07112=1054.318,74.577,421.794,171.203,32.115,156.013
C07113=1054.311,74.327,421.813,171.201,32.113,156.013
C07114=1054.306,74.078,421.830,171.200,32.111,156.012
C07115=1054.300,73.829,421.848,171.198,32.109,156.012
C07116=1054.293,73.579,421.867,171.196,32.106,156.012
C07117=1054.288,73.330,421.884,171.195,32.104,156.011
C07118=1054.282,73.081,421.902,171.193,32.101,156.011
C07119=1054.275,72.832,421.921,171.191,32.099,156.011
C07120=1054.270,72.583,421.939,171.191,32.097,156.010
C07121=1054.264,72.333,421.956,171.189,32.095,156.010
C07122=1054.257,72.084,421.975,171.187,32.092,156.009
C07123=1054.251,71.835,421.992,171.186,32.090,156.009
C07124=1054.245,71.585,422.010,171.184,32.088,156.009
C07125=1054.239,71.335,422.028,171.182,32.085,156.008
C07126=1054.233,71.087,422.046,171.181,32.084,156.008
C07127=1054.227,70.837,422.064,171.179,32.081,156.008
C07128=1054.221,70.588,422.082,171.177,32.079,156.007
C07129=1054.215,70.339,422.100,171.176,32.076,156.007
C07130=1054.208,70.090,422.118,171.174,32.074,156.007
C07131=1054.202,69.841,422.135,171.172,32.072,156.006
C07132=1054.196,69.591,422.153,171.171,32.070,156.006
C07133=1054.190,69.341,422.171,171.170,32.068,156.006
C07134=1054.185,69.092,422.189,171.168,32.065,156.005
C07135=1054.177,68.843,422.207,171.167,32.063,156.005
C07136=1054.171,68.594,422.225,171.165,32.060,156.004
C07137=1054.166,68.345,422.242,171.163,32.058,156.004
C07138=1054.160,68.095,422.260,171.162,32.056,156.004
C07139=1054.153,67.846,422.277,171.160,32.054,156.003
C07140=1054.147,67.596,422.295,171.158,32.052,156.003
C07141=1054.141,67.347,422.313,171.157,32.049,156.003
C07142=1054.135,67.098,422.331,171.155,32.047,156.002
C07143=1054.128,66.849,422.349,171.153,32.045,156.002
C07144=1054.123,66.600,422.366,171.152,32.042,156.002
C07145=1054.117,66.350,422.384,171.151,32.040,156.001
C07146=1054.110,66.101,422.401,171.149,32.038,156.001
C07147=1054.104,65.852,422.419,171.148,32.036,156.001
C07148=1054.098,65.602,422.437,171.146,32.034,156.000
C07149=1054.092,65.353,422.454,171.144,32.031,156.000
C07150=1054.086,65.103,422.472,171.143,32.029,156.000
C07151=1054.080,64.854,422.489,171.141,32.026,155.999
C07152=1054.074,64.605,422.507,171.139,32.024,155.999
C07153=1054.067,64.355,422.525,171.138,32.022,155.999
C07154=1054.062,64.106,422.542,171.136,32.020,155.998
C07155=1054.055,63.857,422.560,171.134,32.018,155.998
C07156=1054.050,63.608,422.577,171.133,32.016,155.998
C07157=1054.043,63.358,422.595,171.132,32.013,155.997
C07158=1054.037,63.108,422.612,171.130,32.011,155.997
C07159=1054.030,62.860,422.629,171.129,32.009,155.997
C07160=1054.023,62.610,422.647,171.127,32.007,155.996
C07161=1054.018,62.361,422.664,171.125,32.004,155.996
C07162=1054.007,61.970,422.692,171.123,32.001,155.995
C07163=1053.998,61.578,422.719,171.120,31.998,155.995
C07164=1053.988,61.187,422.747,171.118,31.994,155.994
C07165=1053.978,60.795,422.774,171.115,31.991,155.994
C07166=1053.972,60.546,422.792,171.114,31.988,155.993
C07167=1053.966,60.296,422.808,171.113,31.986,155.993
C07168=1053.959,60.047,422.825,171.111,31.984,155.993
C07169=1053.953,59.797,422.843,171.109,31.982,155.992
C07170=1053.947,59.549,422.860,171.108,31.980,155.992
C07171=1053.941,59.299,422.878,171.106,31.978,155.992
C07172=1053.935,59.050,422.895,171.104,31.976,155.991
C07173=1053.929,58.801,422.913,171.103,31.973,155.991
C07174=1053.923,58.551,422.929,171.101,31.971,155.991
C07175=1053.916,58.302,422.946,171.099,31.969,155.990
C07176=1053.910,58.053,422.964,171.097,31.967,155.990
C07177=1053.903,57.803,422.981,171.096,31.964,155.990
C07178=1053.894,57.411,423.008,171.094,31.961,155.989
C07179=1053.884,57.018,423.035,171.092,31.958,155.989
C07180=1053.874,56.625,423.063,171.089,31.954,155.988
C07181=1053.865,56.233,423.090,171.086,31.950,155.988
C07182=1053.858,55.984,423.107,171.085,31.948,155.987
C07183=1053.852,55.734,423.124,171.083,31.946,155.987
C07184=1053.846,55.485,423.141,171.081,31.944,155.987
C07185=1053.840,55.235,423.158,171.080,31.942,155.986
C07186=1053.834,54.986,423.176,171.078,31.940,155.986
C07187=1053.828,54.737,423.192,171.077,31.938,155.986
C07188=1053.821,54.487,423.210,171.076,31.935,155.985
C07189=1053.816,54.238,423.227,171.074,31.933,155.985
C07190=1053.809,53.989,423.245,171.072,31.931,155.985
C07191=1053.803,53.740,423.261,171.071,31.928,155.984
C07192=1053.797,53.490,423.279,171.069,31.926,155.984
C07193=1053.790,53.241,423.296,171.067,31.924,155.984
C07194=1053.785,52.992,423.312,171.066,31.922,155.983
C07195=1053.778,52.742,423.330,171.064,31.920,155.983
C07196=1053.772,52.493,423.346,171.062,31.918,155.983
C07197=1053.766,52.243,423.364,171.061,31.915,155.982
C07198=1053.760,51.994,423.381,171.060,31.913,155.982
C07199=1053.754,51.745,423.397,171.058,31.911,155.981
C07200=1053.748,51.495,423.415,171.057,31.908,155.981
C07201=1053.742,51.246,423.432,171.055,31.906,155.981
C07202=1053.736,50.997,423.448,171.053,31.904,155.980
C07203=1053.730,50.747,423.466,171.052,31.902,155.980
C07204=1053.724,50.498,423.483,171.050,31.900,155.980
C07205=1053.717,50.249,423.500,171.048,31.897,155.979
C07206=1053.711,50.000,423.518,171.047,31.895,155.979
C07207=1053.705,49.750,423.534,171.045,31.893,155.979
C07208=1053.699,49.501,423.551,171.043,31.891,155.978
C07209=1053.693,49.251,423.568,171.043,31.888,155.978
C07210=1053.687,49.002,423.585,171.041,31.886,155.978
C07211=1053.681,48.752,423.602,171.039,31.884,155.977
C07212=1053.675,48.503,423.619,171.038,31.882,155.977
C07213=1053.669,48.254,423.635,171.036,31.879,155.977
C07214=1053.662,48.004,423.653,171.034,31.877,155.976
C07215=1053.657,47.755,423.670,171.033,31.875,155.976
C07216=1053.651,47.506,423.687,171.031,31.873,155.976
C07217=1053.645,47.257,423.703,171.029,31.870,155.975
C07218=1053.638,47.007,423.720,171.028,31.868,155.975
C07219=1053.633,46.758,423.737,171.026,31.866,155.975
C07220=1053.626,46.509,423.754,171.025,31.863,155.974
C07221=1053.620,46.259,423.771,171.024,31.861,155.974
C07222=1053.614,45.974,423.790,171.022,31.859,155.973
C07223=1053.607,45.687,423.809,171.020,31.856,155.973
C07224=1053.600,45.402,423.828,171.018,31.853,155.973
C07225=1053.593,45.116,423.848,171.016,31.851,155.972
C07226=1053.587,44.867,423.865,171.014,31.849,155.972
C07227=1053.581,44.618,423.881,171.013,31.847,155.972
C07228=1053.575,44.368,423.899,171.011,31.844,155.971
C07229=1053.569,44.118,423.915,171.010,31.842,155.971
C07230=1053.563,43.870,423.932,171.009,31.840,155.971
C07231=1053.557,43.620,423.948,171.007,31.837,155.970
C07232=1053.551,43.370,423.966,171.005,31.835,155.970
C07233=1053.545,43.121,423.983,171.004,31.833,155.970
C07234=1053.539,42.872,423.999,171.002,31.831,155.969
C07235=1053.532,42.622,424.015,171.000,31.829,155.969
C07236=1053.526,42.373,424.032,170.999,31.827,155.969
C07237=1053.520,42.124,424.049,170.997,31.825,155.968
C07238=1053.514,41.874,424.065,170.995,31.822,155.968
C07239=1053.507,41.624,424.082,170.994,31.820,155.968
C07240=1053.501,41.376,424.098,170.993,31.818,155.967
C07241=1053.495,41.126,424.115,170.991,31.816,155.967
C07242=1053.489,40.877,424.131,170.989,31.814,155.967
C07243=1053.482,40.628,424.148,170.988,31.811,155.966
C07244=1053.476,40.378,424.165,170.986,31.809,155.966
C07245=1053.470,40.129,424.181,170.984,31.807,155.966
C07246=1053.464,39.880,424.197,170.983,31.805,155.965
C07247=1053.459,39.630,424.213,170.981,31.802,155.965
C07248=1053.452,39.381,424.231,170.979,31.800,155.965
C07249=1053.446,39.131,424.247,170.978,31.798,155.964
C07250=1053.440,38.882,424.264,170.977,31.796,155.964
C07251=1053.435,38.632,424.280,170.975,31.794,155.964
C07252=1053.428,38.382,424.297,170.974,31.792,155.963
C07253=1053.422,38.134,424.314,170.972,31.790,155.963
C07254=1053.416,37.884,424.330,170.970,31.787,155.963
C07255=1053.410,37.635,424.346,170.969,31.785,155.962
C07256=1053.403,37.386,424.362,170.967,31.783,155.962
C07257=1053.397,37.136,424.378,170.965,31.781,155.962
C07258=1053.391,36.886,424.395,170.963,31.779,155.961
C07259=1053.385,36.637,424.411,170.962,31.777,155.961
C07260=1053.378,36.388,424.428,170.961,31.775,155.961
C07261=1053.372,36.139,424.444,170.959,31.772,155.960
C07262=1053.366,35.889,424.461,170.958,31.770,155.960
C07263=1053.359,35.640,424.476,170.956,31.768,155.960
C07264=1053.353,35.391,424.493,170.954,31.766,155.960
C07265=1053.347,35.141,424.509,170.953,31.764,155.959
C07266=1053.341,34.892,424.525,170.951,31.762,155.959
C07267=1053.335,34.642,424.542,170.949,31.759,155.958
C07268=1053.328,34.393,424.558,170.947,31.757,155.958
C07269=1053.322,34.143,424.574,170.946,31.755,155.958
C07270=1053.316,33.894,424.590,170.945,31.753,155.958
C07271=1053.310,33.645,424.606,170.943,31.751,155.957
C07272=1053.304,33.395,424.623,170.942,31.749,155.957
C07273=1053.298,33.145,424.639,170.940,31.746,155.957
C07274=1053.291,32.896,424.655,170.938,31.744,155.956
C07275=1053.285,32.647,424.671,170.937,31.742,155.956
C07276=1053.279,32.398,424.687,170.935,31.740,155.956
C07277=1053.273,32.148,424.704,170.933,31.738,155.955
C07278=1053.267,31.899,424.720,170.931,31.736,155.955
C07279=1053.261,31.650,424.736,170.930,31.733,155.955
C07280=1053.254,31.400,424.752,170.929,31.731,155.954
